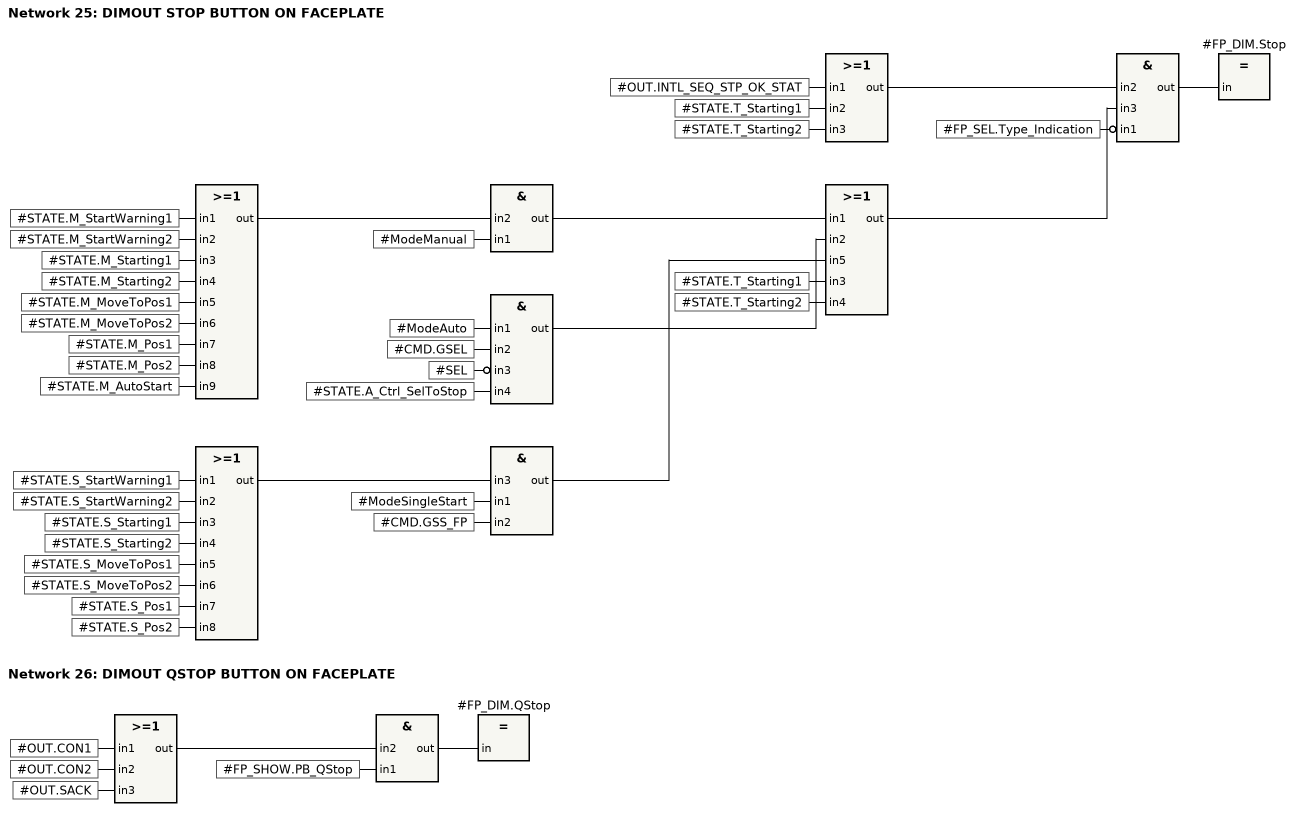
   #FP_DIM.Stop := (#OUT.INTL_SEQ_STP_OK_STAT OR #STATE.T_Starting1 OR #STATE.T_Starting2) AND (((#STATE.M_StartWarning1 OR #STATE.M_StartWarning2 OR #STATE.M_Starting1 OR #STATE.M_Starting2 OR #STATE.M_MoveToPos1 OR #STATE.M_MoveToPos2 OR #STATE.M_Pos1 OR #STATE.M_Pos2 OR #STATE.M_AutoStart) AND #ModeManual) OR (#ModeAuto AND #CMD.GSEL AND NOT #SEL AND #STATE.A_Ctrl_SelToStop) OR ((#STATE.S_StartWarning1 OR #STATE.S_StartWarning2 OR #STATE.S_Starting1 OR #STATE.S_Starting2 OR #STATE.S_MoveToPos1 OR #STATE.S_MoveToPos2 OR #STATE.S_Pos1 OR #STATE.S_Pos2) AND #ModeSingleStart AND #CMD.GSS_FP) OR #STATE.T_Starting1 OR #STATE.T_Starting2) AND NOT #FP_SEL.Type_Indication;
END_REGION

REGION Network 26: DIMOUT QSTOP BUTTON ON FACEPLATE
   #FP_DIM.QStop := (#OUT.CON1 OR #OUT.CON2 OR #OUT.SACK) AND #FP_SHOW.PB_QStop;
END_REGION

REGION Network 27: DIMOUT START1 BUTTON ON FACEPLATE
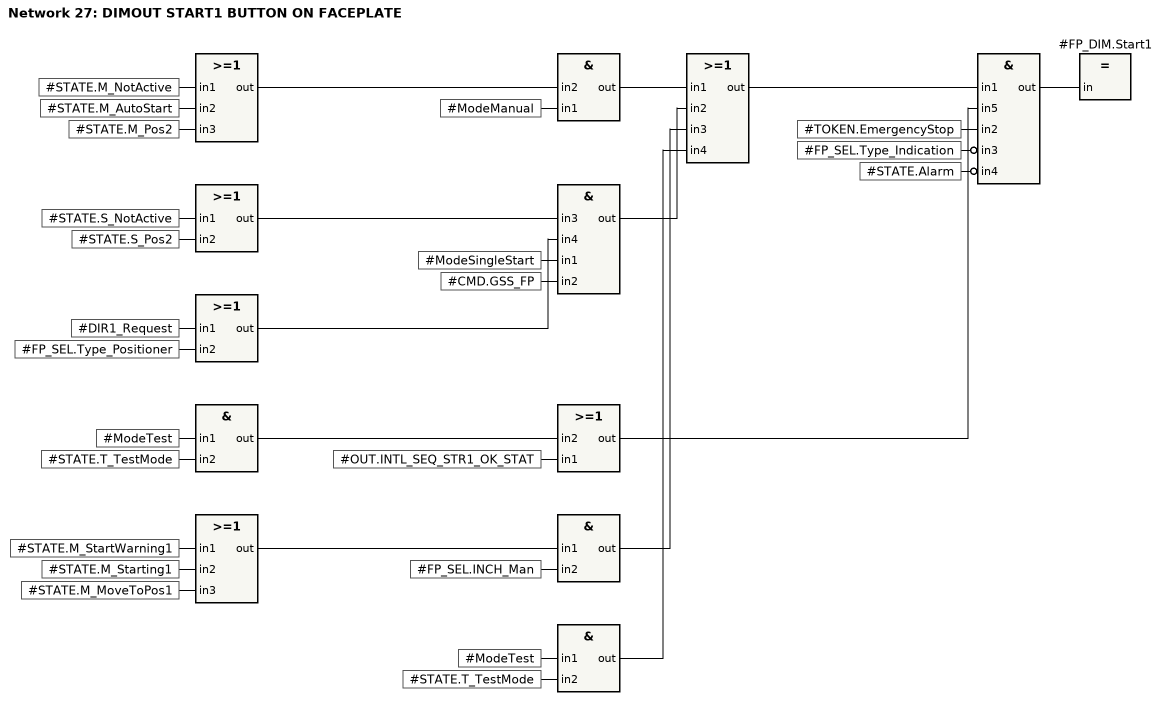
   #FP_DIM.Start1 := (((#STATE.M_NotActive OR #STATE.M_AutoStart OR #STATE.M_Pos2) AND #ModeManual) OR ((#STATE.S_NotActive OR #STATE.S_Pos2) AND (#DIR1_Request OR #FP_SEL.Type_Positioner) AND #ModeSingleStart AND #CMD.GSS_FP) OR ((#STATE.M_StartWarning1 OR #STATE.M_Starting1 OR #STATE.M_MoveToPos1) AND #FP_SEL.INCH_Man) OR (#ModeTest AND #STATE.T_TestMode)) AND ((#ModeTest AND #STATE.T_TestMode) OR #OUT.INTL_SEQ_STR1_OK_STAT) AND #TOKEN.EmergencyStop AND NOT #FP_SEL.Type_Indication AND NOT #STATE.Alarm;
END_REGION

REGION Network 28: DIMOUT START2 BUTTON ON FACEPLATE
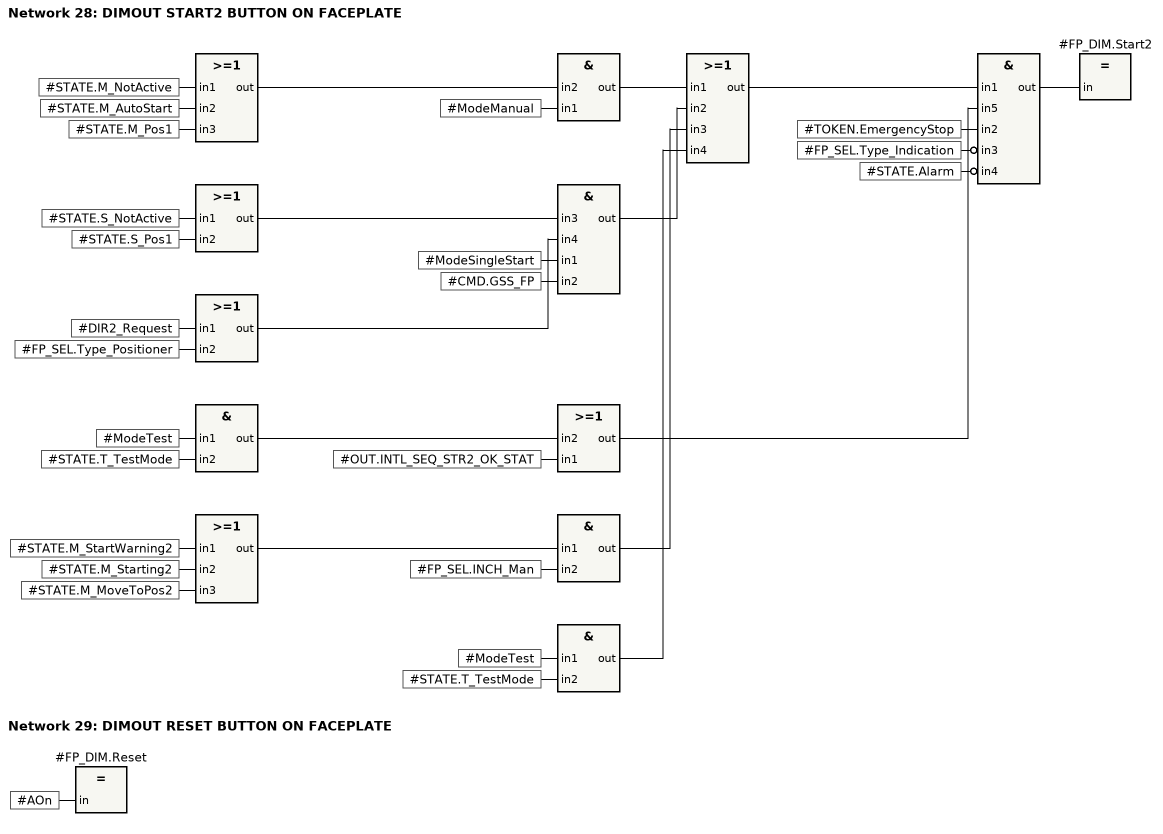
   #FP_DIM.Start2 := (((#STATE.M_NotActive OR #STATE.M_AutoStart OR #STATE.M_Pos1) AND #ModeManual) OR ((#STATE.S_NotActive OR #STATE.S_Pos1) AND (#DIR2_Request OR #FP_SEL.Type_Positioner) AND #ModeSingleStart AND #CMD.GSS_FP) OR ((#STATE.M_StartWarning2 OR #STATE.M_Starting2 OR #STATE.M_MoveToPos2) AND #FP_SEL.INCH_Man) OR (#ModeTest AND #STATE.T_TestMode)) AND ((#ModeTest AND #STATE.T_TestMode) OR #OUT.INTL_SEQ_STR2_OK_STAT) AND #TOKEN.EmergencyStop AND NOT #FP_SEL.Type_Indication AND NOT #STATE.Alarm;
END_REGION

REGION Network 29: DIMOUT RESET BUTTON ON FACEPLATE
   #FP_DIM.Reset := #AOn;
END_REGION

REGION Network 30: Auto Mode
   // Build 002 - 25 March 2019 : REM flag is removed from FP_CMD.Auto condition
   // Build 002 - 25 March 2019 : FP_EN.Mode_Auto flag added to select condition
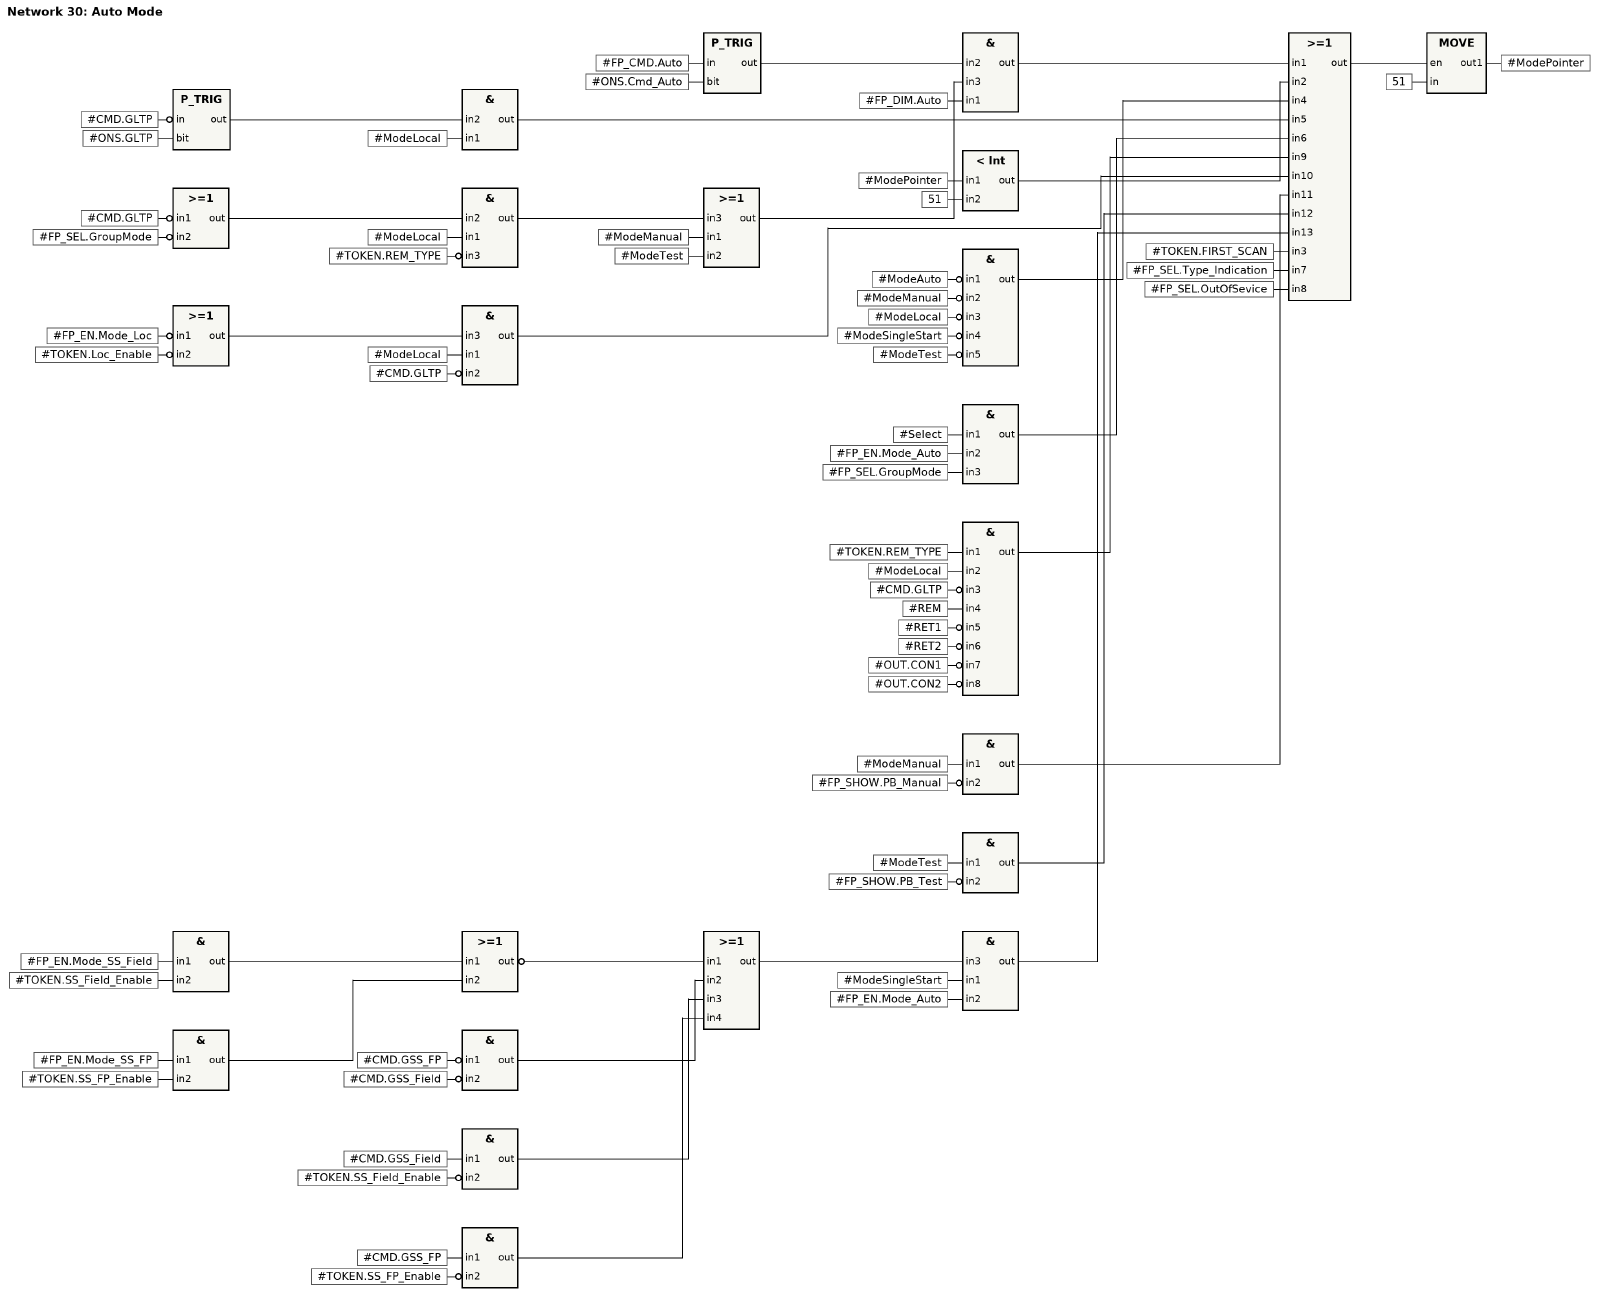
   #_w1 := #FP_CMD.Auto AND NOT #ONS.Cmd_Auto;   // rising edge
   #ONS.Cmd_Auto := #FP_CMD.Auto;
   #_w2 := NOT #CMD.GLTP AND NOT #ONS.GLTP;   // rising edge
   #ONS.GLTP := NOT #CMD.GLTP;
   IF (#_w1 AND (((NOT #CMD.GLTP OR NOT #FP_SEL.GroupMode) AND #ModeLocal AND NOT #TOKEN.REM_TYPE) OR #ModeManual OR #ModeTest) AND #FP_DIM.Auto) OR (#ModePointer < 51) OR (NOT #ModeAuto AND NOT #ModeManual AND NOT #ModeLocal AND NOT #ModeSingleStart AND NOT #ModeTest) OR (#_w2 AND #ModeLocal) OR (#Select AND #FP_EN.Mode_Auto AND #FP_SEL.GroupMode) OR (#TOKEN.REM_TYPE AND #ModeLocal AND NOT #CMD.GLTP AND #REM AND NOT #RET1 AND NOT #RET2 AND NOT #OUT.CON1 AND NOT #OUT.CON2) OR ((NOT #FP_EN.Mode_Loc OR NOT #TOKEN.Loc_Enable) AND #ModeLocal AND NOT #CMD.GLTP) OR (#ModeManual AND NOT #FP_SHOW.PB_Manual) OR (#ModeTest AND NOT #FP_SHOW.PB_Test) OR ((NOT ((#FP_EN.Mode_SS_Field AND #TOKEN.SS_Field_Enable) OR (#FP_EN.Mode_SS_FP AND #TOKEN.SS_FP_Enable)) OR (NOT #CMD.GSS_FP AND NOT #CMD.GSS_Field) OR (#CMD.GSS_Field AND NOT #TOKEN.SS_Field_Enable) OR (#CMD.GSS_FP AND NOT #TOKEN.SS_FP_Enable)) AND #ModeSingleStart AND #FP_EN.Mode_Auto) OR #TOKEN.FIRST_SCAN OR #FP_SEL.Type_Indication OR #FP_SEL.OutOfSevice THEN
       #ModePointer := 51;
   END_IF;
END_REGION

REGION Network 31: Mode Manual
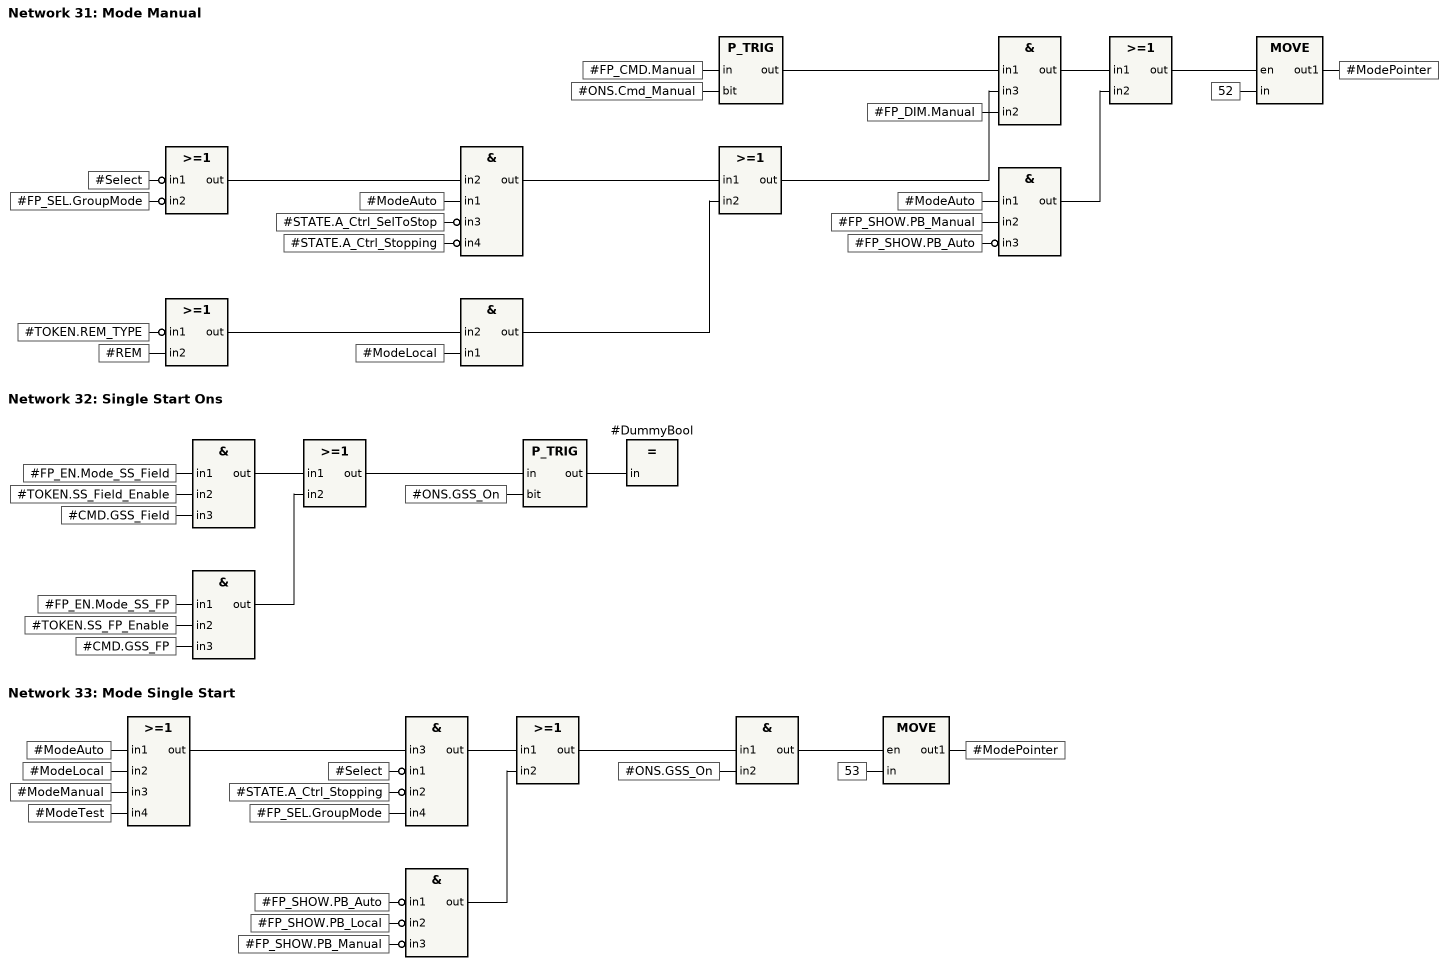
   #_w1 := #FP_CMD.Manual AND NOT #ONS.Cmd_Manual;   // rising edge
   #ONS.Cmd_Manual := #FP_CMD.Manual;
   IF (#_w1 AND (((NOT #Select OR NOT #FP_SEL.GroupMode) AND #ModeAuto AND NOT #STATE.A_Ctrl_SelToStop AND NOT #STATE.A_Ctrl_Stopping) OR ((NOT #TOKEN.REM_TYPE OR #REM) AND #ModeLocal)) AND #FP_DIM.Manual) OR (#ModeAuto AND #FP_SHOW.PB_Manual AND NOT #FP_SHOW.PB_Auto) THEN
       #ModePointer := 52;
   END_IF;
END_REGION

REGION Network 32: Single Start Ons
   // Build 003 - 2.July.2019 (EXTBOB): Added ONS and Created New Network to separate trigger from pre-conditions
   #_w1 := (#FP_EN.Mode_SS_Field AND #TOKEN.SS_Field_Enable AND #CMD.GSS_Field) OR (#FP_EN.Mode_SS_FP AND #TOKEN.SS_FP_Enable AND #CMD.GSS_FP);
   #_w2 := #_w1 AND NOT #ONS.GSS_On;   // rising edge
   #ONS.GSS_On := #_w1;
   #DummyBool := #_w2;
END_REGION

REGION Network 33: Mode Single Start
   // Build 003 - 2.July.2019 (EXTBOB): Added Single Start ONS and Removed the Single start trigger condition & made as seperate Network above
   IF (((#ModeAuto OR #ModeLocal OR #ModeManual OR #ModeTest) AND NOT #Select AND NOT #STATE.A_Ctrl_Stopping AND #FP_SEL.GroupMode) OR (NOT #FP_SHOW.PB_Auto AND NOT #FP_SHOW.PB_Local AND NOT #FP_SHOW.PB_Manual)) AND #ONS.GSS_On THEN
       #ModePointer := 53;
   END_IF;
END_REGION

REGION Network 34: Mode Local
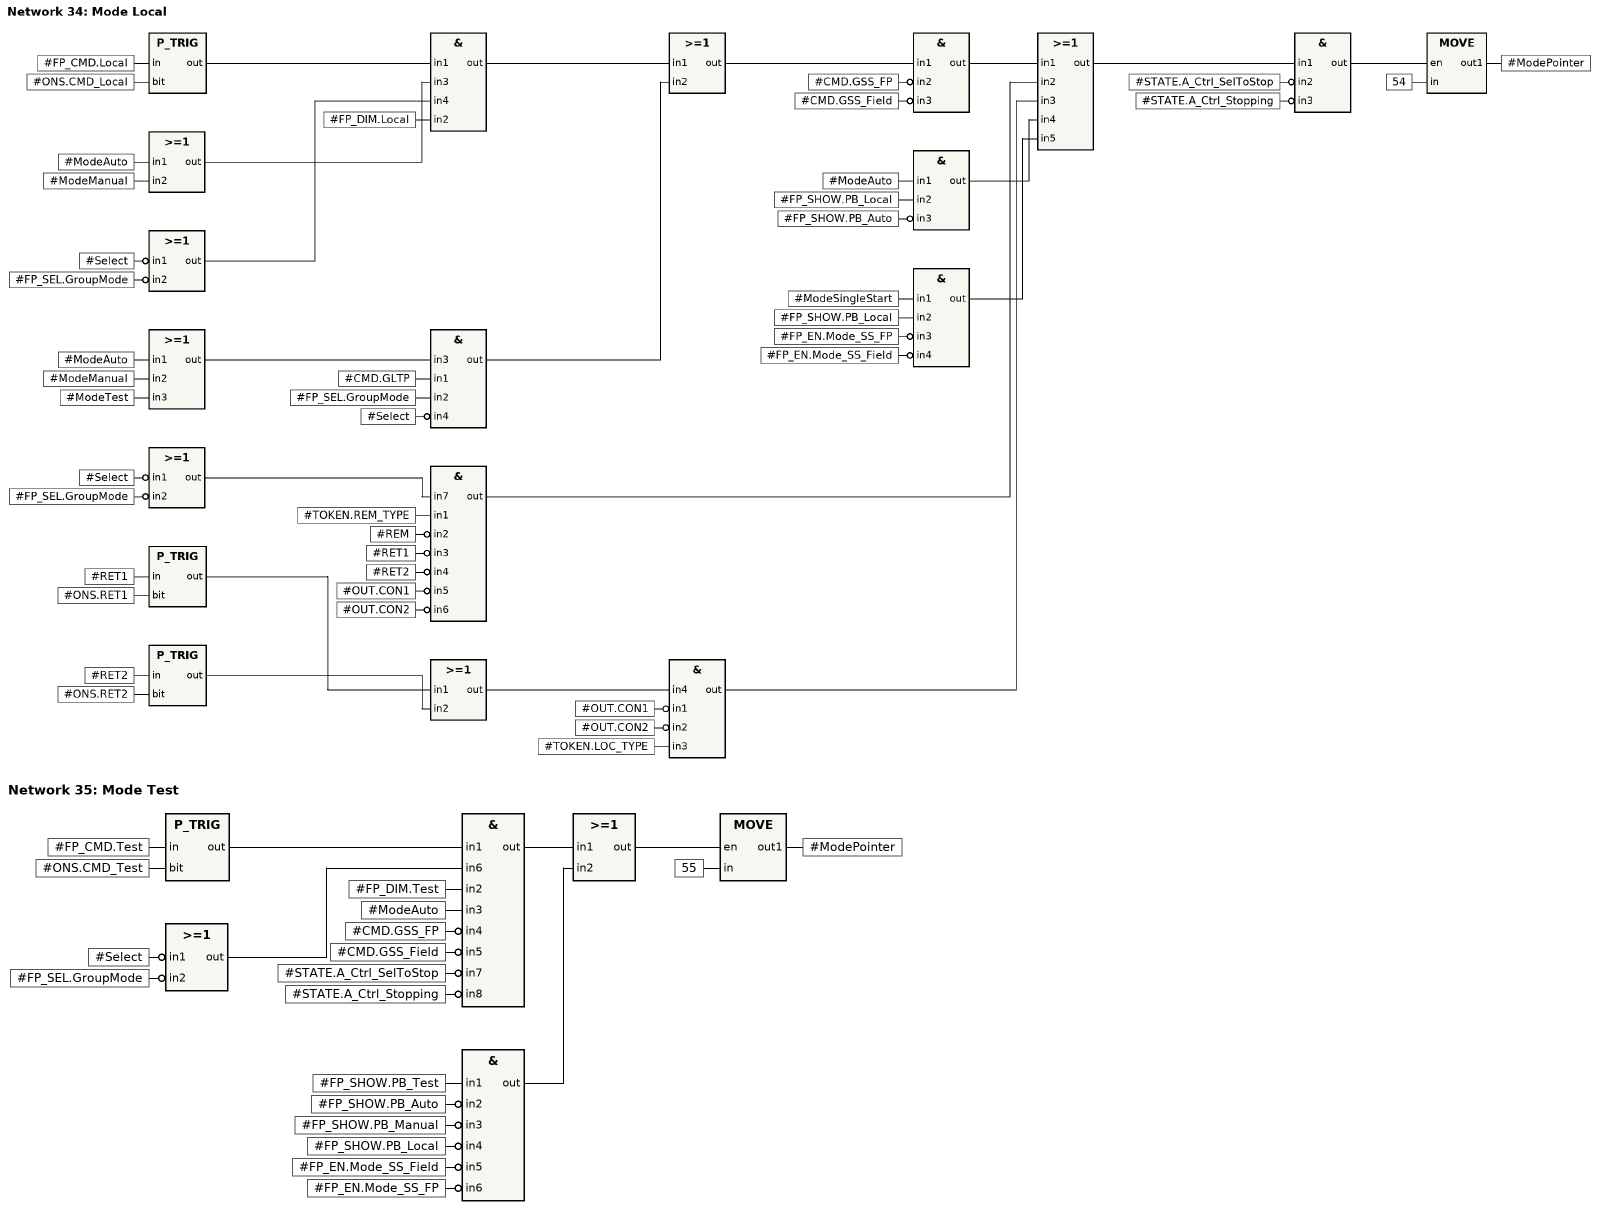
   #_w1 := #FP_CMD.Local AND NOT #ONS.CMD_Local;   // rising edge
   #ONS.CMD_Local := #FP_CMD.Local;
   #_w2 := #RET1 AND NOT #ONS.RET1;   // rising edge
   #ONS.RET1 := #RET1;
   #_w3 := #RET2 AND NOT #ONS.RET2;   // rising edge
   #ONS.RET2 := #RET2;
   IF ((((#_w1 AND (#ModeAuto OR #ModeManual) AND (NOT #Select OR NOT #FP_SEL.GroupMode) AND #FP_DIM.Local) OR ((#ModeAuto OR #ModeManual OR #ModeTest) AND #CMD.GLTP AND #FP_SEL.GroupMode AND NOT #Select)) AND NOT #CMD.GSS_FP AND NOT #CMD.GSS_Field) OR ((NOT #Select OR NOT #FP_SEL.GroupMode) AND #TOKEN.REM_TYPE AND NOT #REM AND NOT #RET1 AND NOT #RET2 AND NOT #OUT.CON1 AND NOT #OUT.CON2) OR ((#_w2 OR #_w3) AND NOT #OUT.CON1 AND NOT #OUT.CON2 AND #TOKEN.LOC_TYPE) OR (#ModeAuto AND #FP_SHOW.PB_Local AND NOT #FP_SHOW.PB_Auto) OR (#ModeSingleStart AND #FP_SHOW.PB_Local AND NOT #FP_EN.Mode_SS_FP AND NOT #FP_EN.Mode_SS_Field)) AND NOT #STATE.A_Ctrl_SelToStop AND NOT #STATE.A_Ctrl_Stopping THEN
       #ModePointer := 54;
   END_IF;
END_REGION

REGION Network 35: Mode Test
   #_w1 := #FP_CMD.Test AND NOT #ONS.CMD_Test;   // rising edge
   #ONS.CMD_Test := #FP_CMD.Test;
   IF (#_w1 AND (NOT #Select OR NOT #FP_SEL.GroupMode) AND #FP_DIM.Test AND #ModeAuto AND NOT #CMD.GSS_FP AND NOT #CMD.GSS_Field AND NOT #STATE.A_Ctrl_SelToStop AND NOT #STATE.A_Ctrl_Stopping) OR (#FP_SHOW.PB_Test AND NOT #FP_SHOW.PB_Auto AND NOT #FP_SHOW.PB_Manual AND NOT #FP_SHOW.PB_Local AND NOT #FP_EN.Mode_SS_Field AND NOT #FP_EN.Mode_SS_FP) THEN
       #ModePointer := 55;
   END_IF;
END_REGION

REGION Network 36: Mode Auto
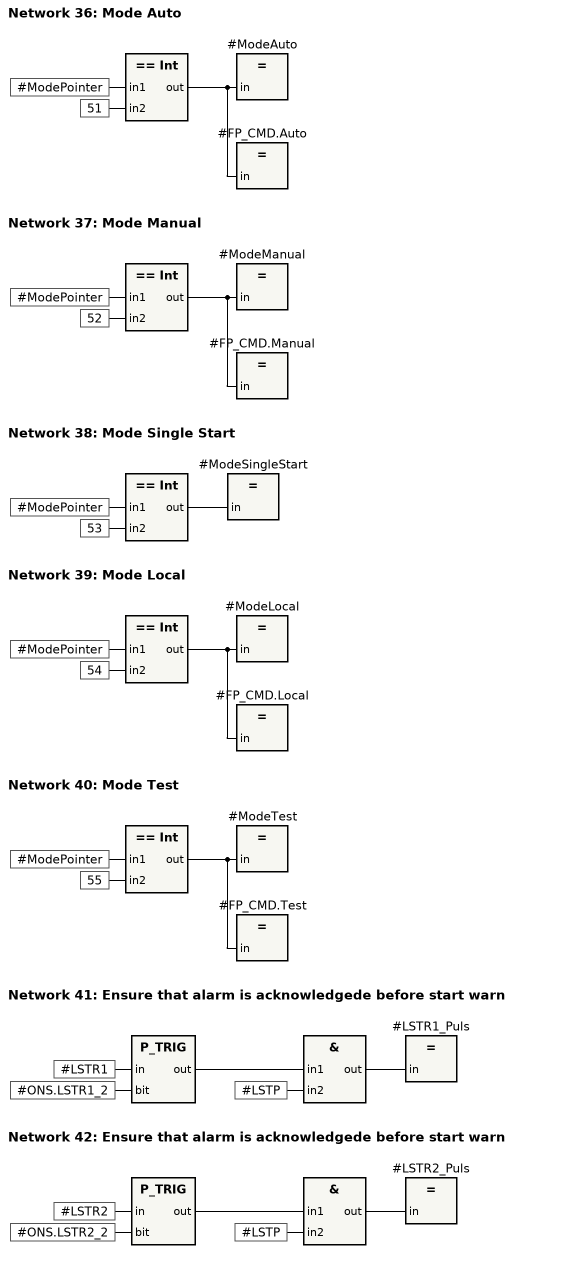
   #ModeAuto := #ModePointer = 51;
   #FP_CMD.Auto := #ModeAuto;
END_REGION

REGION Network 37: Mode Manual
   #ModeManual := #ModePointer = 52;
   #FP_CMD.Manual := #ModeManual;
END_REGION

REGION Network 38: Mode Single Start
   #ModeSingleStart := #ModePointer = 53;
END_REGION

REGION Network 39: Mode Local
   #ModeLocal := #ModePointer = 54;
   #FP_CMD.Local := #ModeLocal;
END_REGION

REGION Network 40: Mode Test
   #ModeTest := #ModePointer = 55;
   #FP_CMD.Test := #ModeTest;
END_REGION

REGION Network 41: Ensure that alarm is acknowledgede before start warn
   // Build 003 - 30 June 2019 (EXTBOB): Added LSTP to prevent pulse output
   #_w1 := #LSTR1 AND NOT #ONS.LSTR1_2;   // rising edge
   #ONS.LSTR1_2 := #LSTR1;
   #LSTR1_Puls := #_w1 AND #LSTP;
END_REGION

REGION Network 42: Ensure that alarm is acknowledgede before start warn
   // Build 003 - 30 June 2019 (EXTBOB): Added LSTP to prevent pulse output
   #_w1 := #LSTR2 AND NOT #ONS.LSTR2_2;   // rising edge
   #ONS.LSTR2_2 := #LSTR2;
   #LSTR2_Puls := #_w1 AND #LSTP;
END_REGION

REGION Network 43: FACEPLATE COMMANDS (Pulse Type)
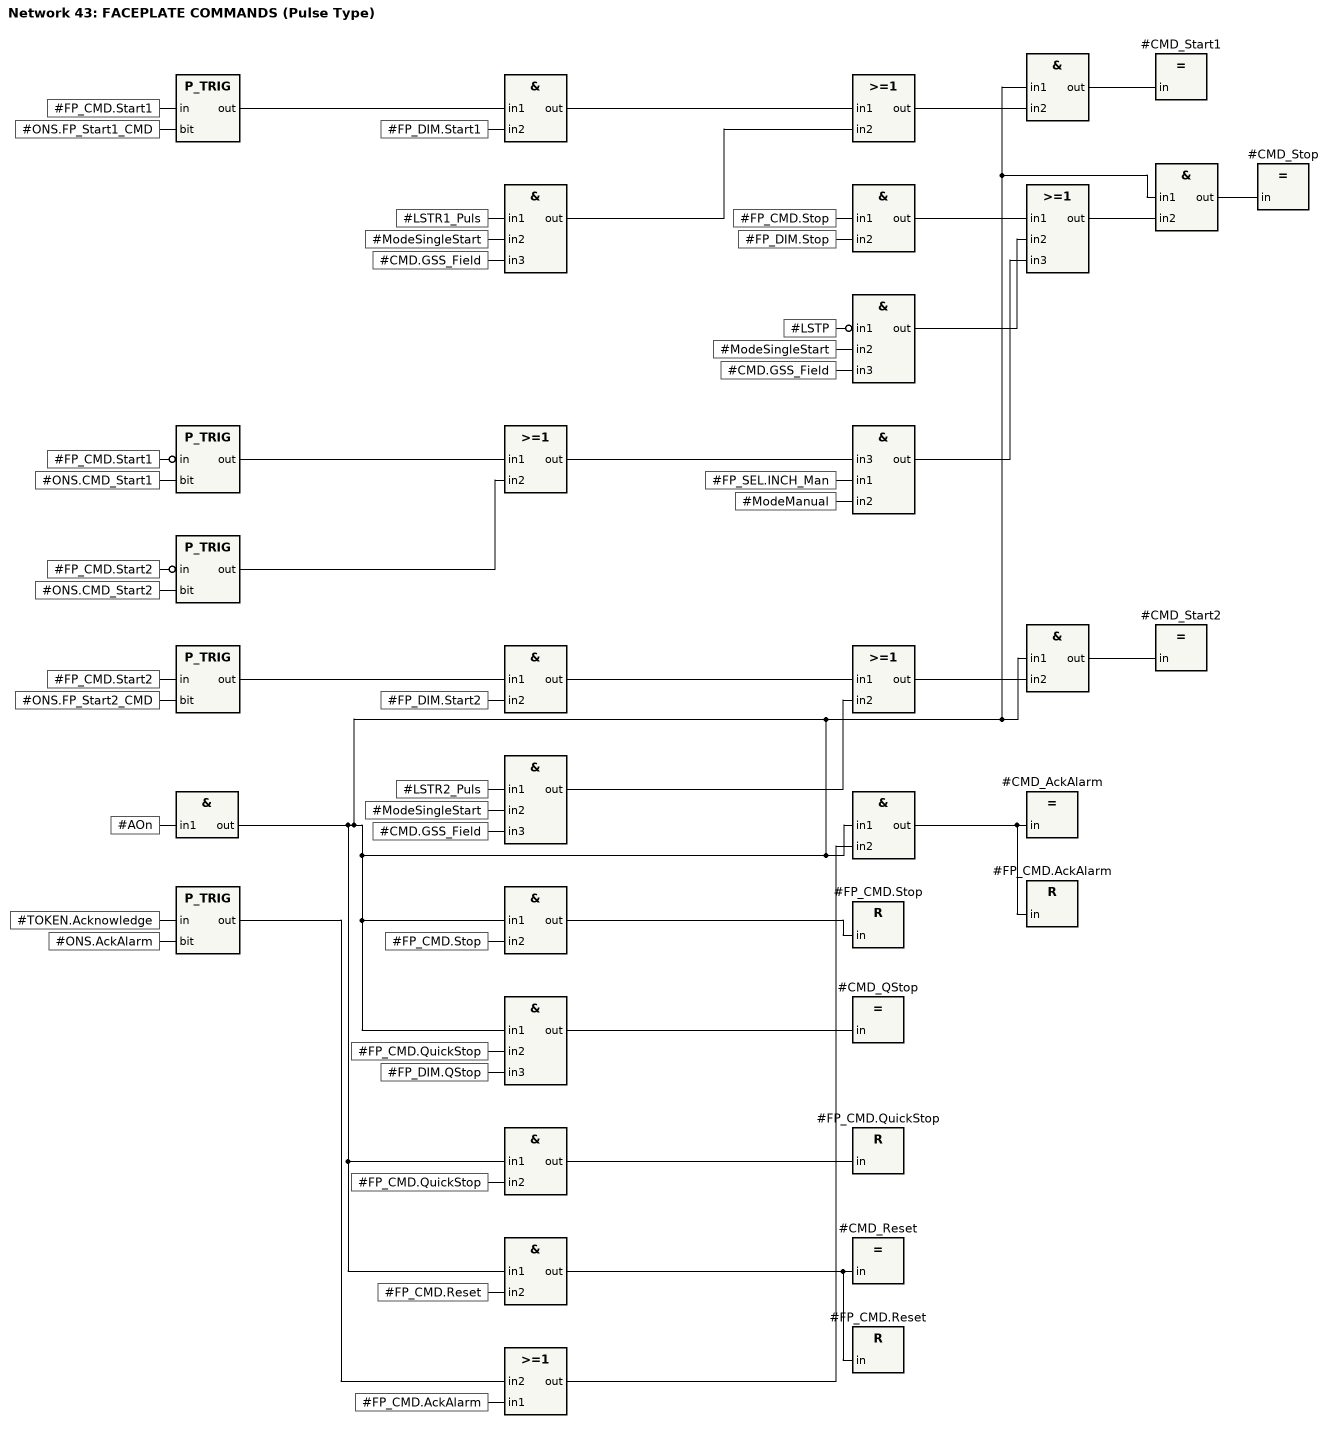
   #_w1 := #FP_CMD.Start1 AND NOT #ONS.FP_Start1_CMD;   // rising edge
   #ONS.FP_Start1_CMD := #FP_CMD.Start1;
   #CMD_Start1 := #AOn AND ((#_w1 AND #FP_DIM.Start1) OR (#LSTR1_Puls AND #ModeSingleStart AND #CMD.GSS_Field));
   #_w2 := #FP_CMD.Start2 AND NOT #ONS.FP_Start2_CMD;   // rising edge
   #ONS.FP_Start2_CMD := #FP_CMD.Start2;
   #CMD_Start2 := #AOn AND ((#_w2 AND #FP_DIM.Start2) OR (#LSTR2_Puls AND #ModeSingleStart AND #CMD.GSS_Field));
   #_w3 := NOT #FP_CMD.Start1 AND NOT #ONS.CMD_Start1;   // rising edge
   #ONS.CMD_Start1 := NOT #FP_CMD.Start1;
   #_w4 := NOT #FP_CMD.Start2 AND NOT #ONS.CMD_Start2;   // rising edge
   #ONS.CMD_Start2 := NOT #FP_CMD.Start2;
   #CMD_Stop := #AOn AND ((#FP_CMD.Stop AND #FP_DIM.Stop) OR (NOT #LSTP AND #ModeSingleStart AND #CMD.GSS_Field) OR ((#_w3 OR #_w4) AND #FP_SEL.INCH_Man AND #ModeManual));
   IF #AOn AND #FP_CMD.Stop THEN #FP_CMD.Stop := FALSE; END_IF;
   #CMD_QStop := #AOn AND #FP_CMD.QuickStop AND #FP_DIM.QStop;
   IF #AOn AND #FP_CMD.QuickStop THEN #FP_CMD.QuickStop := FALSE; END_IF;
   #CMD_Reset := #AOn AND #FP_CMD.Reset;
   IF #CMD_Reset THEN #FP_CMD.Reset := FALSE; END_IF;
   #_w5 := #TOKEN.Acknowledge AND NOT #ONS.AckAlarm;   // rising edge
   #ONS.AckAlarm := #TOKEN.Acknowledge;
   #CMD_AckAlarm := #AOn AND (#_w5 OR #FP_CMD.AckAlarm);
   IF #CMD_AckAlarm THEN #FP_CMD.AckAlarm := FALSE; END_IF;
END_REGION

REGION Network 44: FACEPLATE COMMANDS (Pulse Type)
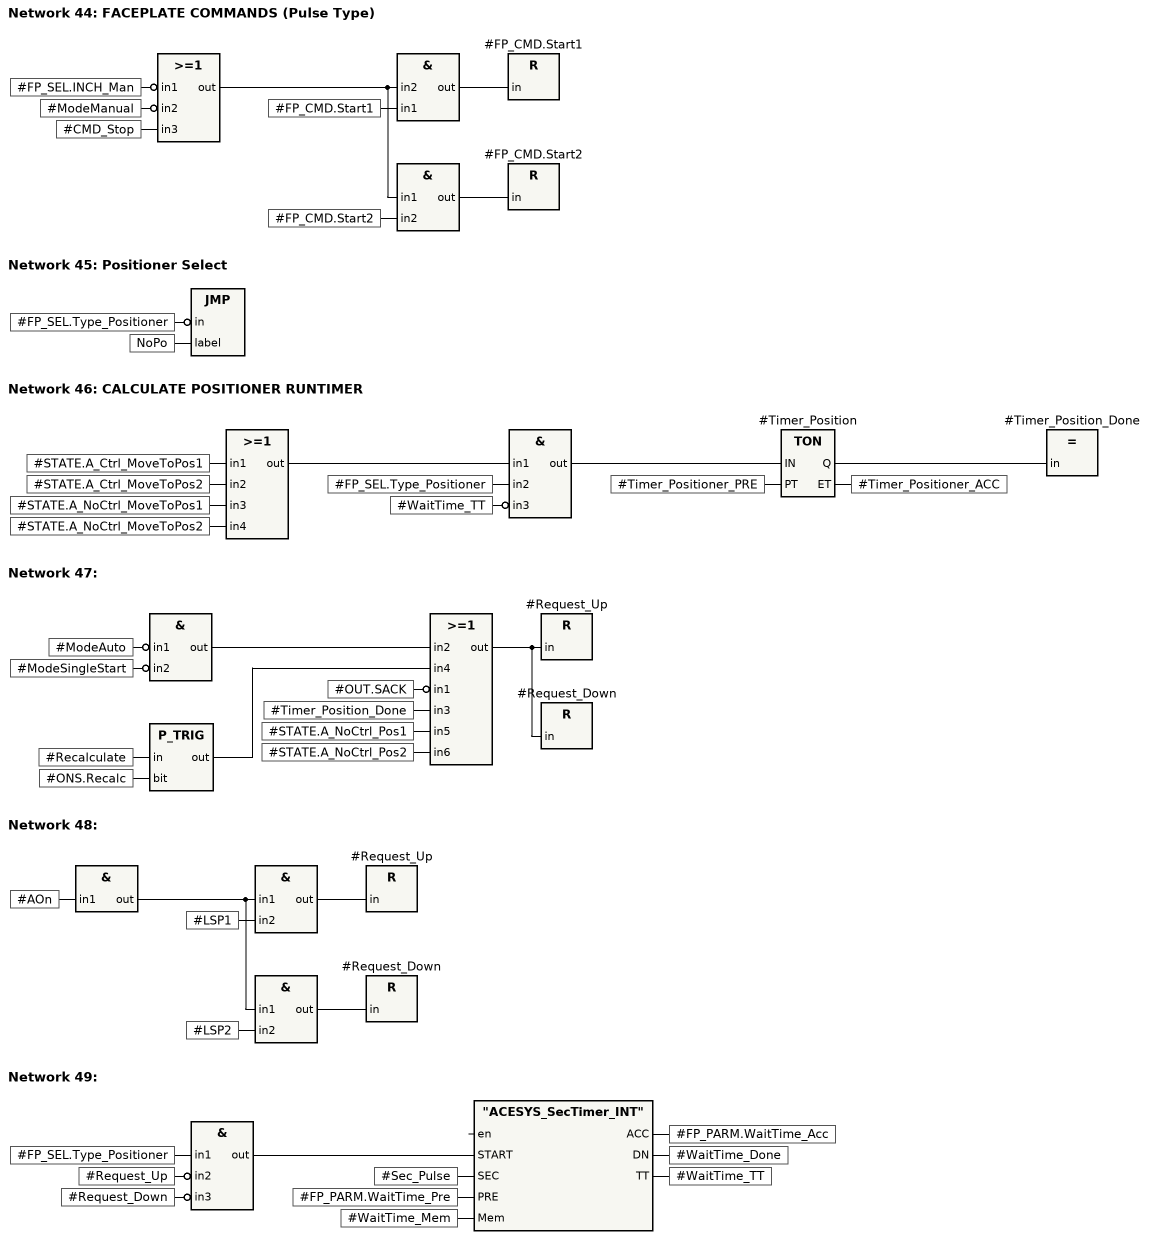
   #_w1 := NOT #FP_SEL.INCH_Man OR NOT #ModeManual OR #CMD_Stop;
   IF #_w1 AND #FP_CMD.Start1 THEN #FP_CMD.Start1 := FALSE; END_IF;
   IF #_w1 AND #FP_CMD.Start2 THEN #FP_CMD.Start2 := FALSE; END_IF;
END_REGION

REGION Network 45: Positioner Select
   IF NOT #FP_SEL.Type_Positioner THEN GOTO NoPo; END_IF;
END_REGION

REGION Network 46: CALCULATE POSITIONER RUNTIMER
   #Timer_Position(IN := (#STATE.A_Ctrl_MoveToPos1 OR #STATE.A_Ctrl_MoveToPos2 OR #STATE.A_NoCtrl_MoveToPos1 OR #STATE.A_NoCtrl_MoveToPos2) AND #FP_SEL.Type_Positioner AND NOT #WaitTime_TT,   // TON
                   PT := #Timer_Positioner_PRE,
                   ET => #Timer_Positioner_ACC);
   #Timer_Position_Done := #Timer_Position.Q;
END_REGION

REGION Network 47
   #_w1 := #Recalculate AND NOT #ONS.Recalc;   // rising edge
   #ONS.Recalc := #Recalculate;
   IF (NOT #ModeAuto AND NOT #ModeSingleStart) OR #_w1 OR NOT #OUT.SACK OR #Timer_Position_Done OR #STATE.A_NoCtrl_Pos1 OR #STATE.A_NoCtrl_Pos2 THEN
       #Request_Up := FALSE;
       #Request_Down := FALSE;
   END_IF;
END_REGION

REGION Network 48
   IF #AOn AND #LSP1 THEN #Request_Up := FALSE; END_IF;
   IF #AOn AND #LSP2 THEN #Request_Down := FALSE; END_IF;
END_REGION

REGION Network 49
   "ACESYS_SecTimer_INT"(START := #FP_SEL.Type_Positioner AND NOT #Request_Up AND NOT #Request_Down,
                         SEC := #Sec_Pulse,
                         PRE := #FP_PARM.WaitTime_Pre,
                         Mem := #WaitTime_Mem,
                         ACC => #FP_PARM.WaitTime_Acc,
                         DN => #WaitTime_Done,
                         TT => #WaitTime_TT);
END_REGION

REGION Network 50
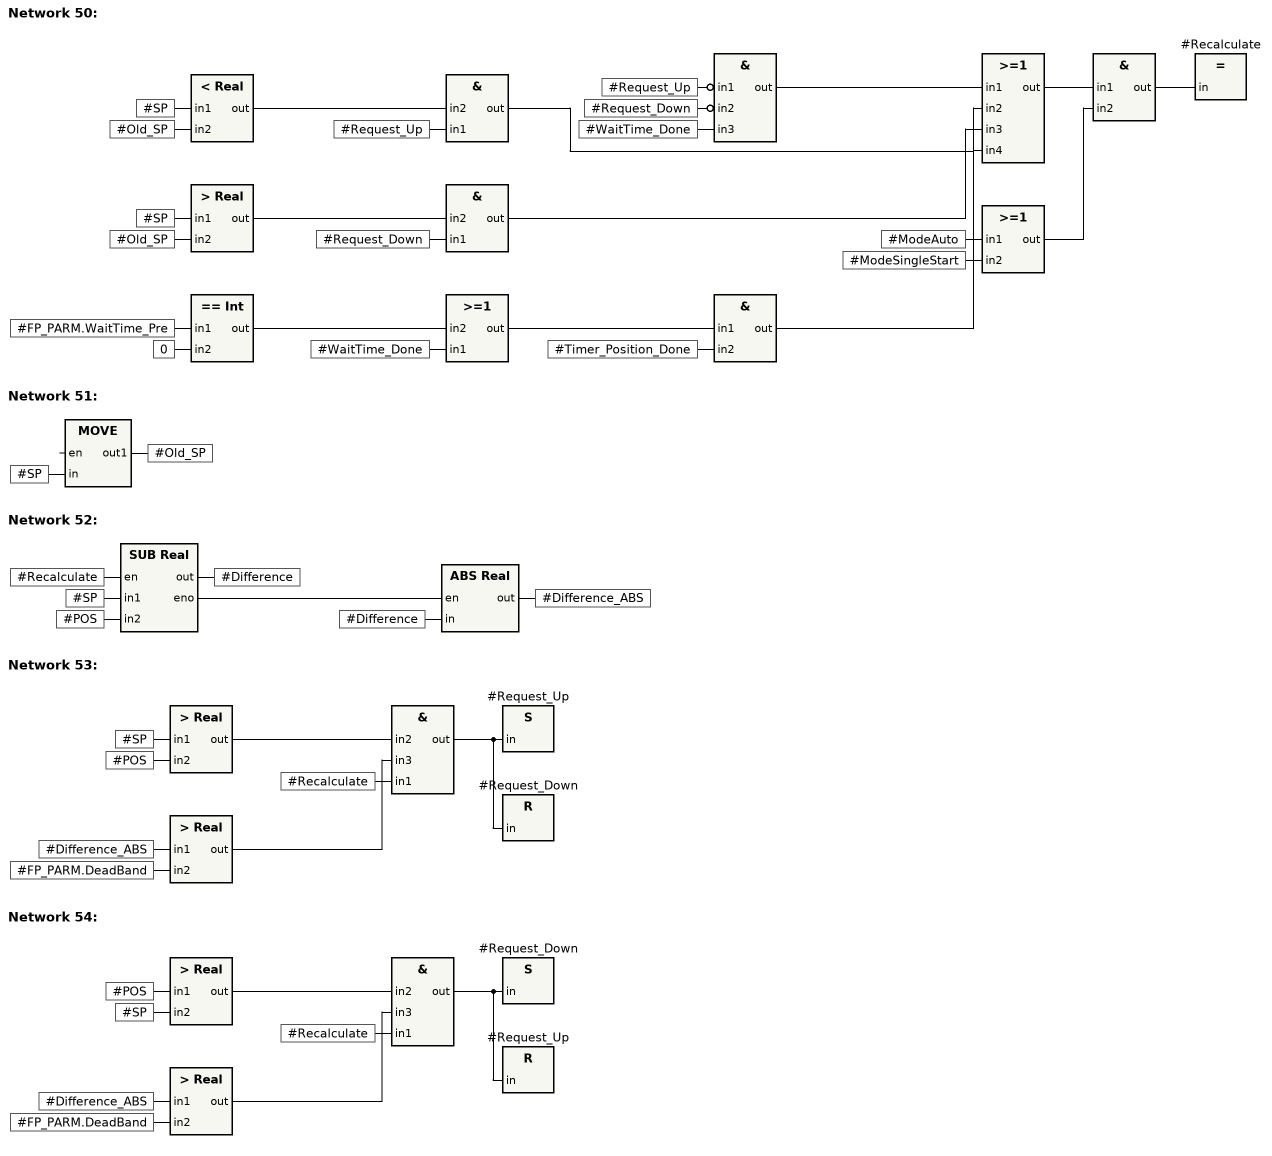
   #Recalculate := ((NOT #Request_Up AND NOT #Request_Down AND #WaitTime_Done) OR ((#SP < #Old_SP) AND #Request_Up) OR ((#SP > #Old_SP) AND #Request_Down) OR (((#FP_PARM.WaitTime_Pre = 0) OR #WaitTime_Done) AND #Timer_Position_Done)) AND (#ModeAuto OR #ModeSingleStart);
END_REGION

REGION Network 51
   #Old_SP := #SP;
END_REGION

REGION Network 52
   // ENO of a box is taken as its EN; it also drops when the box reports an error
   IF #Recalculate THEN
       #Difference := #SP - #POS;
       #Difference_ABS := ABS(#Difference);
   END_IF;
END_REGION

REGION Network 53
   IF (#SP > #POS) AND (#Difference_ABS > #FP_PARM.DeadBand) AND #Recalculate THEN
       #Request_Up := TRUE;
       #Request_Down := FALSE;
   END_IF;
END_REGION

REGION Network 54
   IF (#POS > #SP) AND (#Difference_ABS > #FP_PARM.DeadBand) AND #Recalculate THEN
       #Request_Down := TRUE;
       #Request_Up := FALSE;
   END_IF;
END_REGION

REGION Network 55
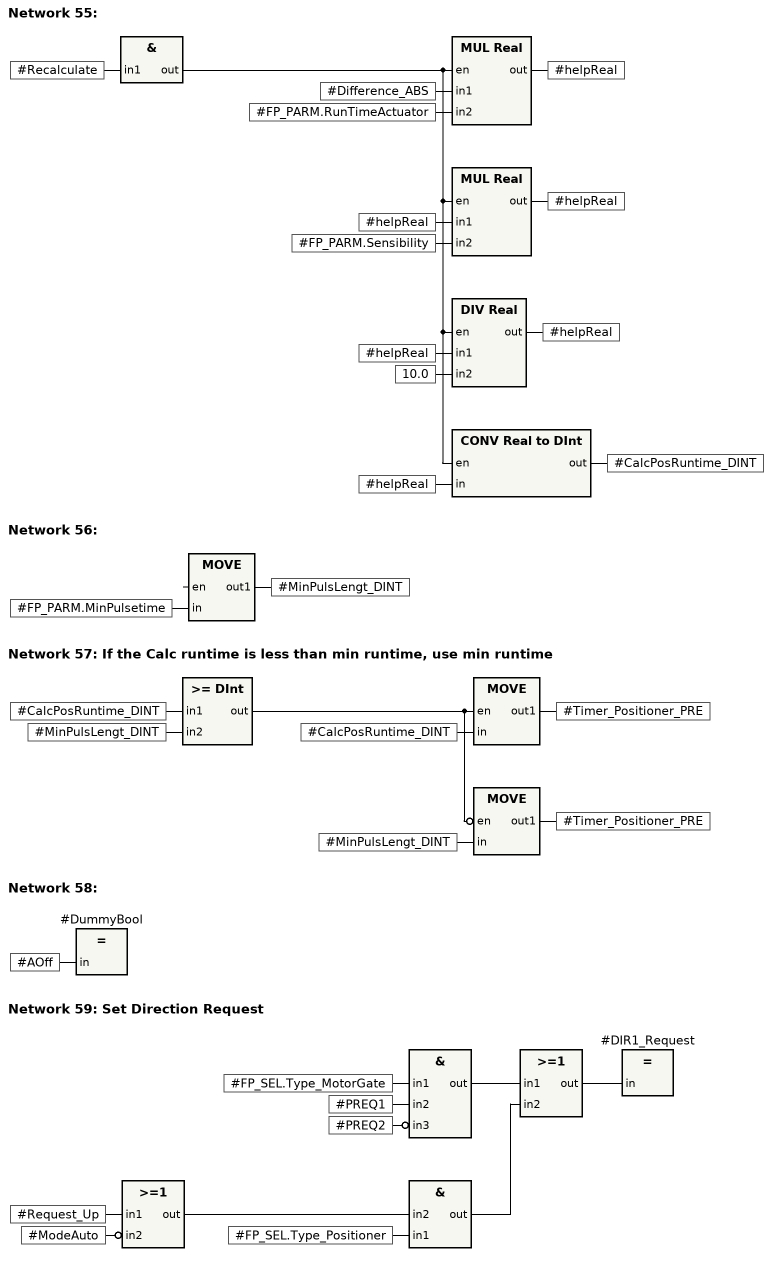
   IF #Recalculate THEN
       #helpReal := #Difference_ABS * #FP_PARM.RunTimeActuator;
       #helpReal := #helpReal * #FP_PARM.Sensibility;
       #helpReal := #helpReal / 10.0;
       #CalcPosRuntime_DINT := REAL_TO_DINT(#helpReal);
   END_IF;
END_REGION

REGION Network 56
   #MinPulsLengt_DINT := #FP_PARM.MinPulsetime;
END_REGION

REGION Network 57: If the Calc runtime is less than min runtime, use min runtime
   #_w1 := #CalcPosRuntime_DINT >= #MinPulsLengt_DINT;
   IF #_w1 THEN #Timer_Positioner_PRE := #CalcPosRuntime_DINT; END_IF;
   IF NOT #_w1 THEN #Timer_Positioner_PRE := #MinPulsLengt_DINT; END_IF;
END_REGION

REGION Network 58
   NoPo:
   #DummyBool := #AOff;
END_REGION

REGION Network 59: Set Direction Request
   #DIR1_Request := (#FP_SEL.Type_MotorGate AND #PREQ1 AND NOT #PREQ2) OR ((#Request_Up OR NOT #ModeAuto) AND #FP_SEL.Type_Positioner);
END_REGION

REGION Network 60
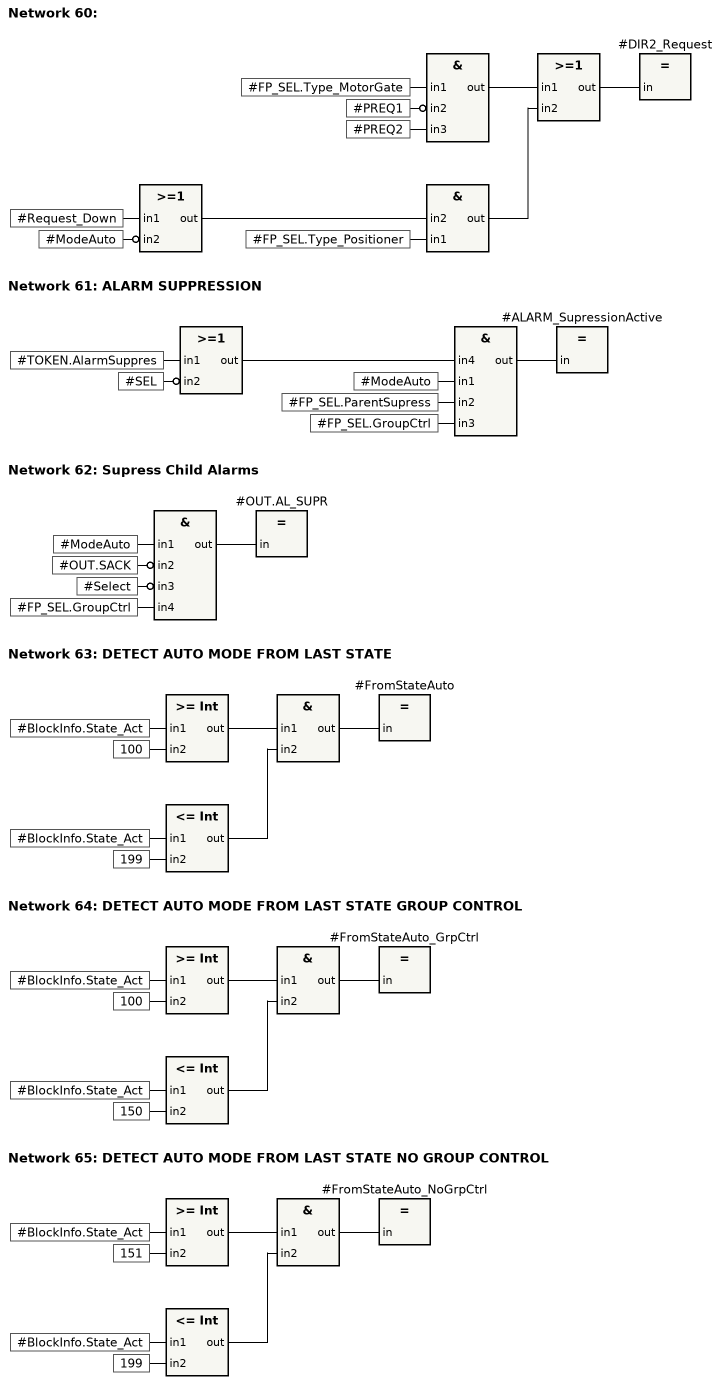
   #DIR2_Request := (#FP_SEL.Type_MotorGate AND NOT #PREQ1 AND #PREQ2) OR ((#Request_Down OR NOT #ModeAuto) AND #FP_SEL.Type_Positioner);
END_REGION

REGION Network 61: ALARM SUPPRESSION
   #ALARM_SupressionActive := (#TOKEN.AlarmSuppres OR NOT #SEL) AND #ModeAuto AND #FP_SEL.ParentSupress AND #FP_SEL.GroupCtrl;
END_REGION

REGION Network 62: Supress Child Alarms
   #OUT.AL_SUPR := #ModeAuto AND NOT #OUT.SACK AND NOT #Select AND #FP_SEL.GroupCtrl;
END_REGION

REGION Network 63: DETECT AUTO MODE FROM LAST STATE
   #FromStateAuto := (#BlockInfo.State_Act >= 100) AND (#BlockInfo.State_Act <= 199);
END_REGION

REGION Network 64: DETECT AUTO MODE FROM LAST STATE GROUP CONTROL
   #FromStateAuto_GrpCtrl := (#BlockInfo.State_Act >= 100) AND (#BlockInfo.State_Act <= 150);
END_REGION

REGION Network 65: DETECT AUTO MODE FROM LAST STATE NO GROUP CONTROL
   #FromStateAuto_NoGrpCtrl := (#BlockInfo.State_Act >= 151) AND (#BlockInfo.State_Act <= 199);
END_REGION

REGION Network 66: DETECT SS MODE FROM LAST STATE
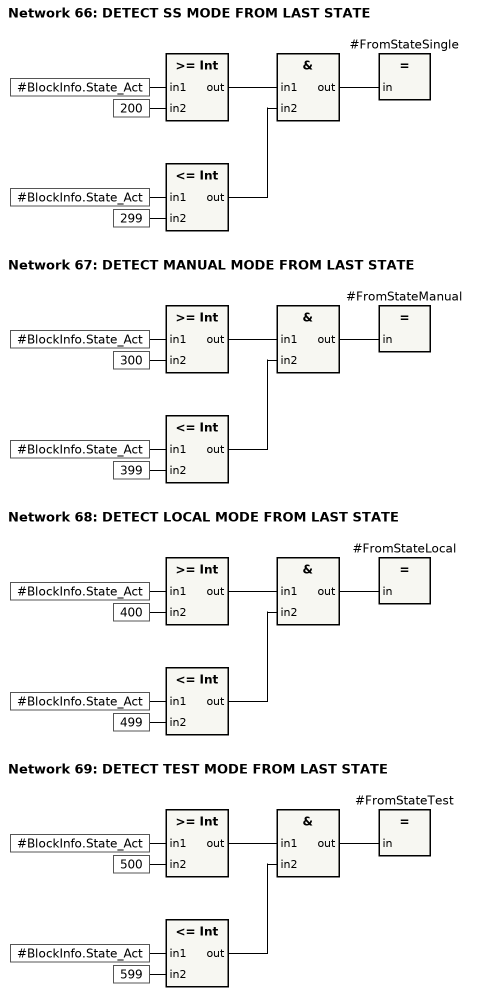
   #FromStateSingle := (#BlockInfo.State_Act >= 200) AND (#BlockInfo.State_Act <= 299);
END_REGION

REGION Network 67: DETECT MANUAL MODE FROM LAST STATE
   #FromStateManual := (#BlockInfo.State_Act >= 300) AND (#BlockInfo.State_Act <= 399);
END_REGION

REGION Network 68: DETECT LOCAL MODE FROM LAST STATE
   #FromStateLocal := (#BlockInfo.State_Act >= 400) AND (#BlockInfo.State_Act <= 499);
END_REGION

REGION Network 69: DETECT TEST MODE FROM LAST STATE
   #FromStateTest := (#BlockInfo.State_Act >= 500) AND (#BlockInfo.State_Act <= 599);
END_REGION

REGION Network 70: DETECT MODE FROM LAST STATE - STOP STATE
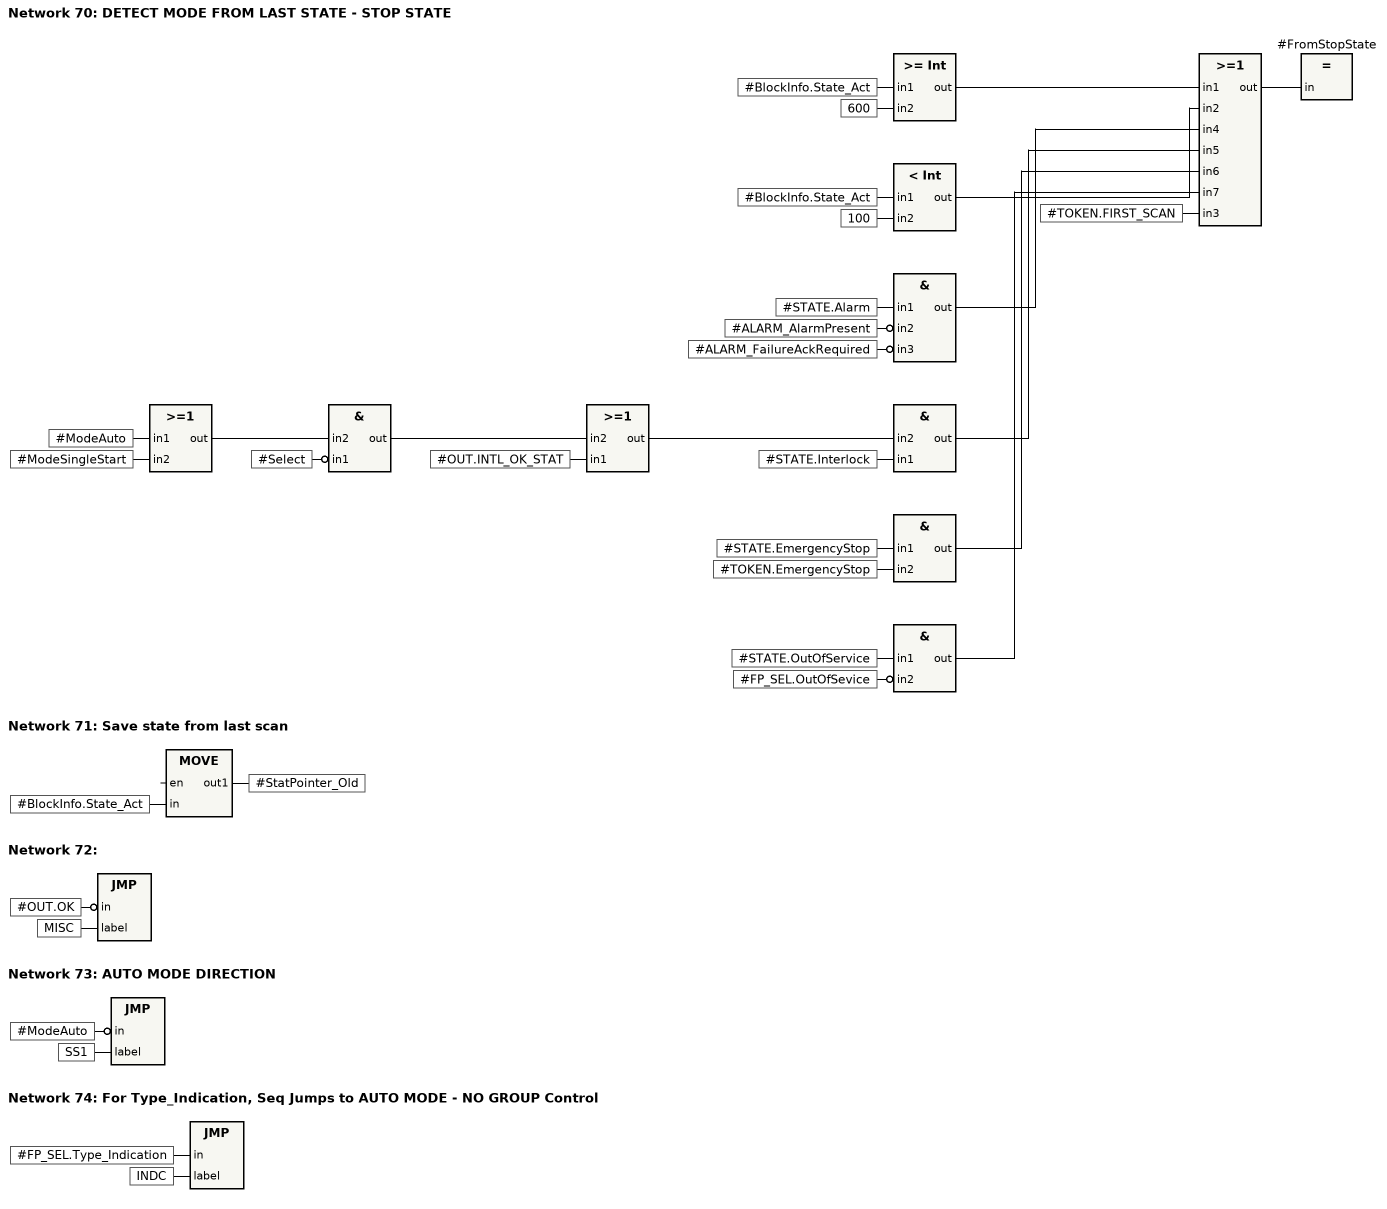
   #FromStopState := (#BlockInfo.State_Act >= 600) OR (#BlockInfo.State_Act < 100) OR (#STATE.Alarm AND NOT #ALARM_AlarmPresent AND NOT #ALARM_FailureAckRequired) OR ((((#ModeAuto OR #ModeSingleStart) AND NOT #Select) OR #OUT.INTL_OK_STAT) AND #STATE.Interlock) OR (#STATE.EmergencyStop AND #TOKEN.EmergencyStop) OR (#STATE.OutOfService AND NOT #FP_SEL.OutOfSevice) OR #TOKEN.FIRST_SCAN;
END_REGION

REGION Network 71: Save state from last scan
   #StatPointer_Old := #BlockInfo.State_Act;
END_REGION

REGION Network 72
   IF NOT #OUT.OK THEN GOTO MISC; END_IF;
END_REGION

REGION Network 73: AUTO MODE DIRECTION
   IF NOT #ModeAuto THEN GOTO SS1; END_IF;
END_REGION

REGION Network 74: For Type_Indication, Seq Jumps to AUTO MODE - NO GROUP Control
   IF #FP_SEL.Type_Indication THEN GOTO INDC; END_IF;
END_REGION

REGION Network 75: AUTO MODE - GROUP CONTROL - State: Auto - Stopped
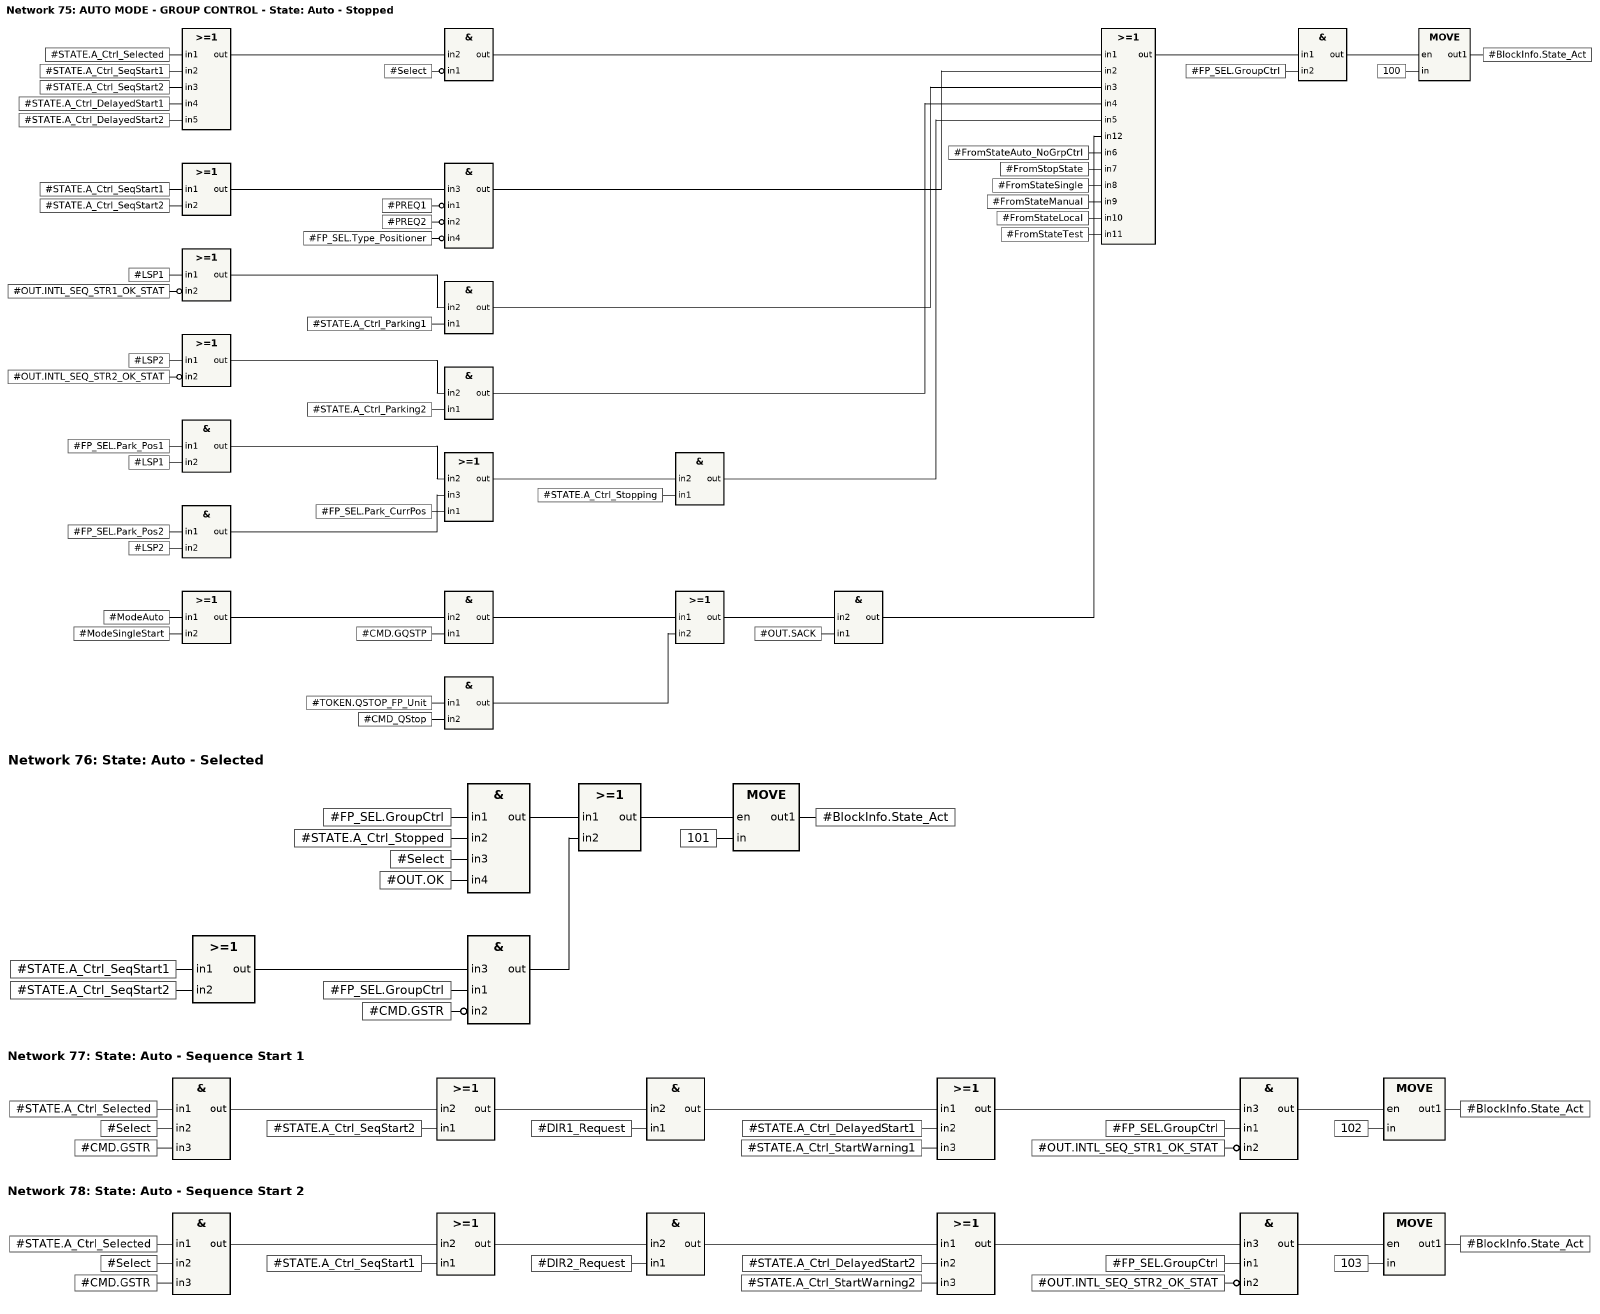
   IF (((#STATE.A_Ctrl_Selected OR #STATE.A_Ctrl_SeqStart1 OR #STATE.A_Ctrl_SeqStart2 OR #STATE.A_Ctrl_DelayedStart1 OR #STATE.A_Ctrl_DelayedStart2) AND NOT #Select) OR ((#STATE.A_Ctrl_SeqStart1 OR #STATE.A_Ctrl_SeqStart2) AND NOT #PREQ1 AND NOT #PREQ2 AND NOT #FP_SEL.Type_Positioner) OR ((#LSP1 OR NOT #OUT.INTL_SEQ_STR1_OK_STAT) AND #STATE.A_Ctrl_Parking1) OR ((#LSP2 OR NOT #OUT.INTL_SEQ_STR2_OK_STAT) AND #STATE.A_Ctrl_Parking2) OR (((#FP_SEL.Park_Pos1 AND #LSP1) OR (#FP_SEL.Park_Pos2 AND #LSP2) OR #FP_SEL.Park_CurrPos) AND #STATE.A_Ctrl_Stopping) OR ((((#ModeAuto OR #ModeSingleStart) AND #CMD.GQSTP) OR (#TOKEN.QSTOP_FP_Unit AND #CMD_QStop)) AND #OUT.SACK) OR #FromStateAuto_NoGrpCtrl OR #FromStopState OR #FromStateSingle OR #FromStateManual OR #FromStateLocal OR #FromStateTest) AND #FP_SEL.GroupCtrl THEN
       #BlockInfo.State_Act := 100;
   END_IF;
END_REGION

REGION Network 76: State: Auto - Selected
   IF (#FP_SEL.GroupCtrl AND #STATE.A_Ctrl_Stopped AND #Select AND #OUT.OK) OR ((#STATE.A_Ctrl_SeqStart1 OR #STATE.A_Ctrl_SeqStart2) AND #FP_SEL.GroupCtrl AND NOT #CMD.GSTR) THEN
       #BlockInfo.State_Act := 101;
   END_IF;
END_REGION

REGION Network 77: State: Auto - Sequence Start 1
   IF ((((#STATE.A_Ctrl_Selected AND #Select AND #CMD.GSTR) OR #STATE.A_Ctrl_SeqStart2) AND #DIR1_Request) OR #STATE.A_Ctrl_DelayedStart1 OR #STATE.A_Ctrl_StartWarning1) AND #FP_SEL.GroupCtrl AND NOT #OUT.INTL_SEQ_STR1_OK_STAT THEN
       #BlockInfo.State_Act := 102;
   END_IF;
END_REGION

REGION Network 78: State: Auto - Sequence Start 2
   IF ((((#STATE.A_Ctrl_Selected AND #Select AND #CMD.GSTR) OR #STATE.A_Ctrl_SeqStart1) AND #DIR2_Request) OR #STATE.A_Ctrl_DelayedStart2 OR #STATE.A_Ctrl_StartWarning2) AND #FP_SEL.GroupCtrl AND NOT #OUT.INTL_SEQ_STR2_OK_STAT THEN
       #BlockInfo.State_Act := 103;
   END_IF;
END_REGION

REGION Network 79: State: Auto - Delayed Start 1
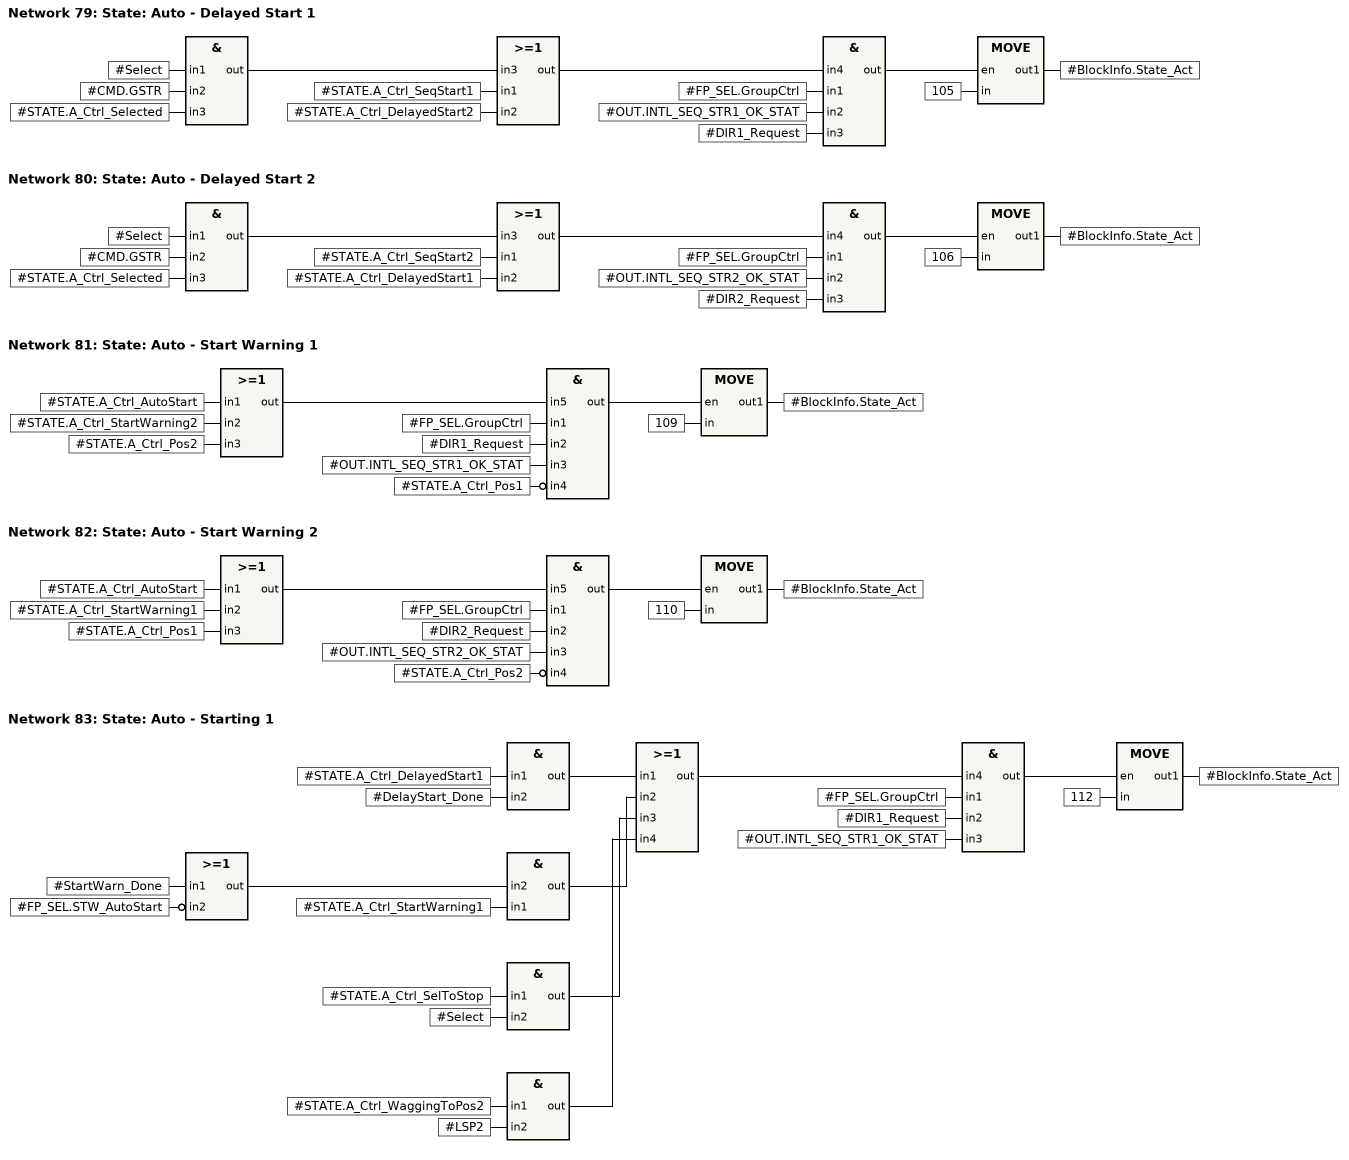
   IF ((#Select AND #CMD.GSTR AND #STATE.A_Ctrl_Selected) OR #STATE.A_Ctrl_SeqStart1 OR #STATE.A_Ctrl_DelayedStart2) AND #FP_SEL.GroupCtrl AND #OUT.INTL_SEQ_STR1_OK_STAT AND #DIR1_Request THEN
       #BlockInfo.State_Act := 105;
   END_IF;
END_REGION

REGION Network 80: State: Auto - Delayed Start 2
   IF ((#Select AND #CMD.GSTR AND #STATE.A_Ctrl_Selected) OR #STATE.A_Ctrl_SeqStart2 OR #STATE.A_Ctrl_DelayedStart1) AND #FP_SEL.GroupCtrl AND #OUT.INTL_SEQ_STR2_OK_STAT AND #DIR2_Request THEN
       #BlockInfo.State_Act := 106;
   END_IF;
END_REGION

REGION Network 81: State: Auto - Start Warning 1
   IF (#STATE.A_Ctrl_AutoStart OR #STATE.A_Ctrl_StartWarning2 OR #STATE.A_Ctrl_Pos2) AND #FP_SEL.GroupCtrl AND #DIR1_Request AND #OUT.INTL_SEQ_STR1_OK_STAT AND NOT #STATE.A_Ctrl_Pos1 THEN
       #BlockInfo.State_Act := 109;
   END_IF;
END_REGION

REGION Network 82: State: Auto - Start Warning 2
   IF (#STATE.A_Ctrl_AutoStart OR #STATE.A_Ctrl_StartWarning1 OR #STATE.A_Ctrl_Pos1) AND #FP_SEL.GroupCtrl AND #DIR2_Request AND #OUT.INTL_SEQ_STR2_OK_STAT AND NOT #STATE.A_Ctrl_Pos2 THEN
       #BlockInfo.State_Act := 110;
   END_IF;
END_REGION

REGION Network 83: State: Auto - Starting 1
   IF ((#STATE.A_Ctrl_DelayedStart1 AND #DelayStart_Done) OR ((#StartWarn_Done OR NOT #FP_SEL.STW_AutoStart) AND #STATE.A_Ctrl_StartWarning1) OR (#STATE.A_Ctrl_SelToStop AND #Select) OR (#STATE.A_Ctrl_WaggingToPos2 AND #LSP2)) AND #FP_SEL.GroupCtrl AND #DIR1_Request AND #OUT.INTL_SEQ_STR1_OK_STAT THEN
       #BlockInfo.State_Act := 112;
   END_IF;
END_REGION

REGION Network 84: state: Auto - Starting 2
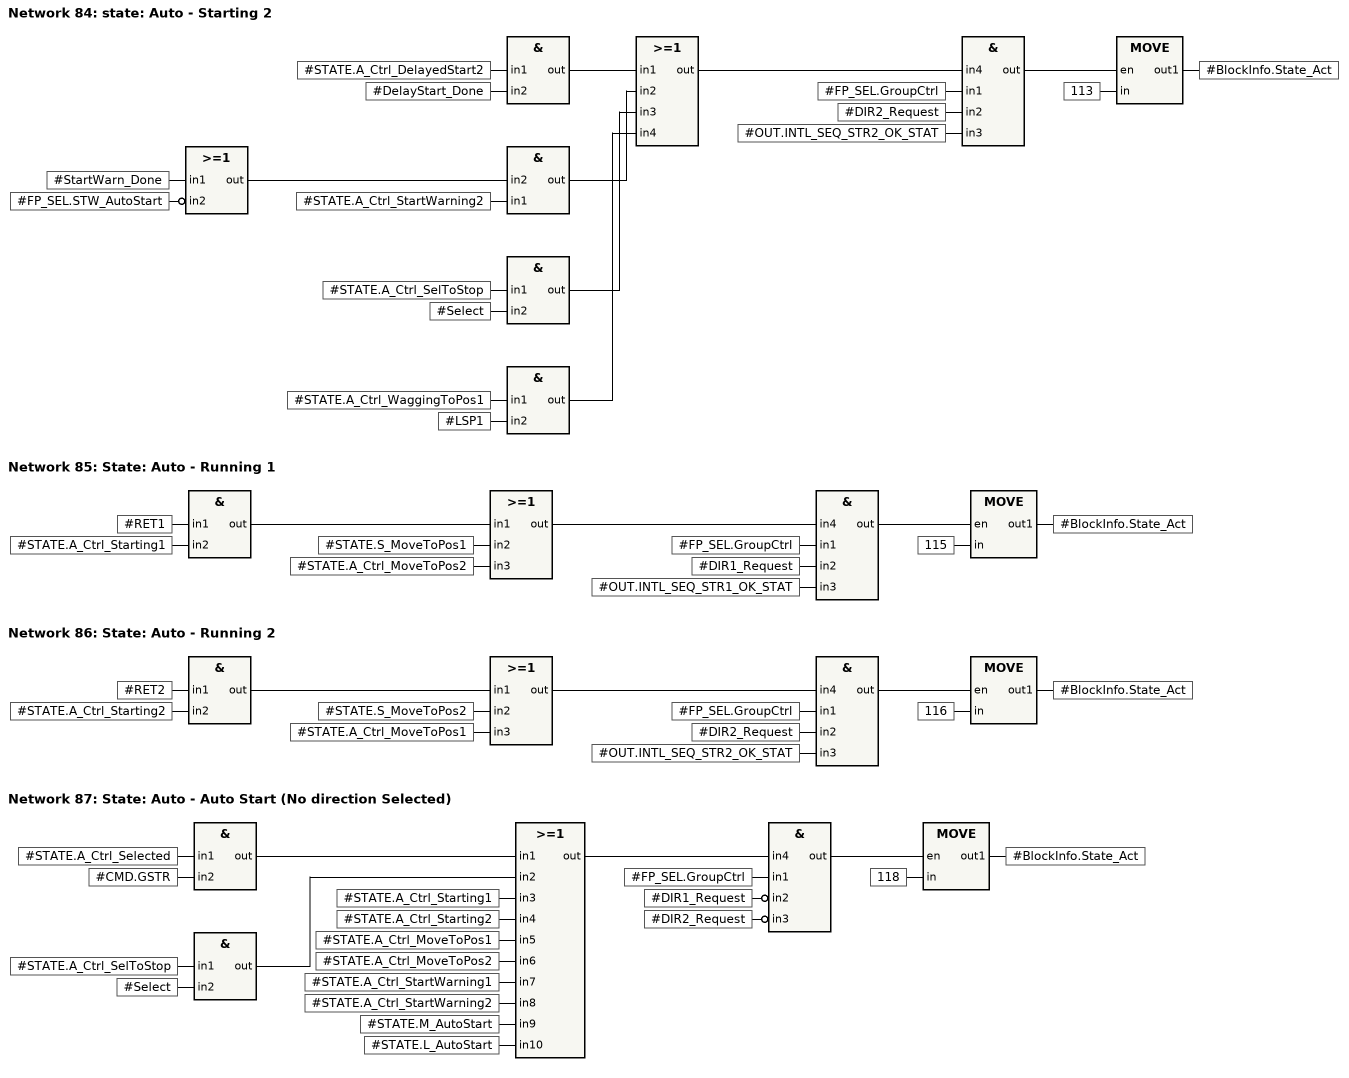
   IF ((#STATE.A_Ctrl_DelayedStart2 AND #DelayStart_Done) OR ((#StartWarn_Done OR NOT #FP_SEL.STW_AutoStart) AND #STATE.A_Ctrl_StartWarning2) OR (#STATE.A_Ctrl_SelToStop AND #Select) OR (#STATE.A_Ctrl_WaggingToPos1 AND #LSP1)) AND #FP_SEL.GroupCtrl AND #DIR2_Request AND #OUT.INTL_SEQ_STR2_OK_STAT THEN
       #BlockInfo.State_Act := 113;
   END_IF;
END_REGION

REGION Network 85: State: Auto - Running 1
   IF ((#RET1 AND #STATE.A_Ctrl_Starting1) OR #STATE.S_MoveToPos1 OR #STATE.A_Ctrl_MoveToPos2) AND #FP_SEL.GroupCtrl AND #DIR1_Request AND #OUT.INTL_SEQ_STR1_OK_STAT THEN
       #BlockInfo.State_Act := 115;
   END_IF;
END_REGION

REGION Network 86: State: Auto - Running 2
   IF ((#RET2 AND #STATE.A_Ctrl_Starting2) OR #STATE.S_MoveToPos2 OR #STATE.A_Ctrl_MoveToPos1) AND #FP_SEL.GroupCtrl AND #DIR2_Request AND #OUT.INTL_SEQ_STR2_OK_STAT THEN
       #BlockInfo.State_Act := 116;
   END_IF;
END_REGION

REGION Network 87: State: Auto - Auto Start (No direction Selected)
   // Build 002 - 26 March 2019 : SetToStop with Select condition is added
   IF ((#STATE.A_Ctrl_Selected AND #CMD.GSTR) OR (#STATE.A_Ctrl_SelToStop AND #Select) OR #STATE.A_Ctrl_Starting1 OR #STATE.A_Ctrl_Starting2 OR #STATE.A_Ctrl_MoveToPos1 OR #STATE.A_Ctrl_MoveToPos2 OR #STATE.A_Ctrl_StartWarning1 OR #STATE.A_Ctrl_StartWarning2 OR #STATE.M_AutoStart OR #STATE.L_AutoStart) AND #FP_SEL.GroupCtrl AND NOT #DIR1_Request AND NOT #DIR2_Request THEN
       #BlockInfo.State_Act := 118;
   END_IF;
END_REGION

REGION Network 88: State: Auto - In Pos. 1
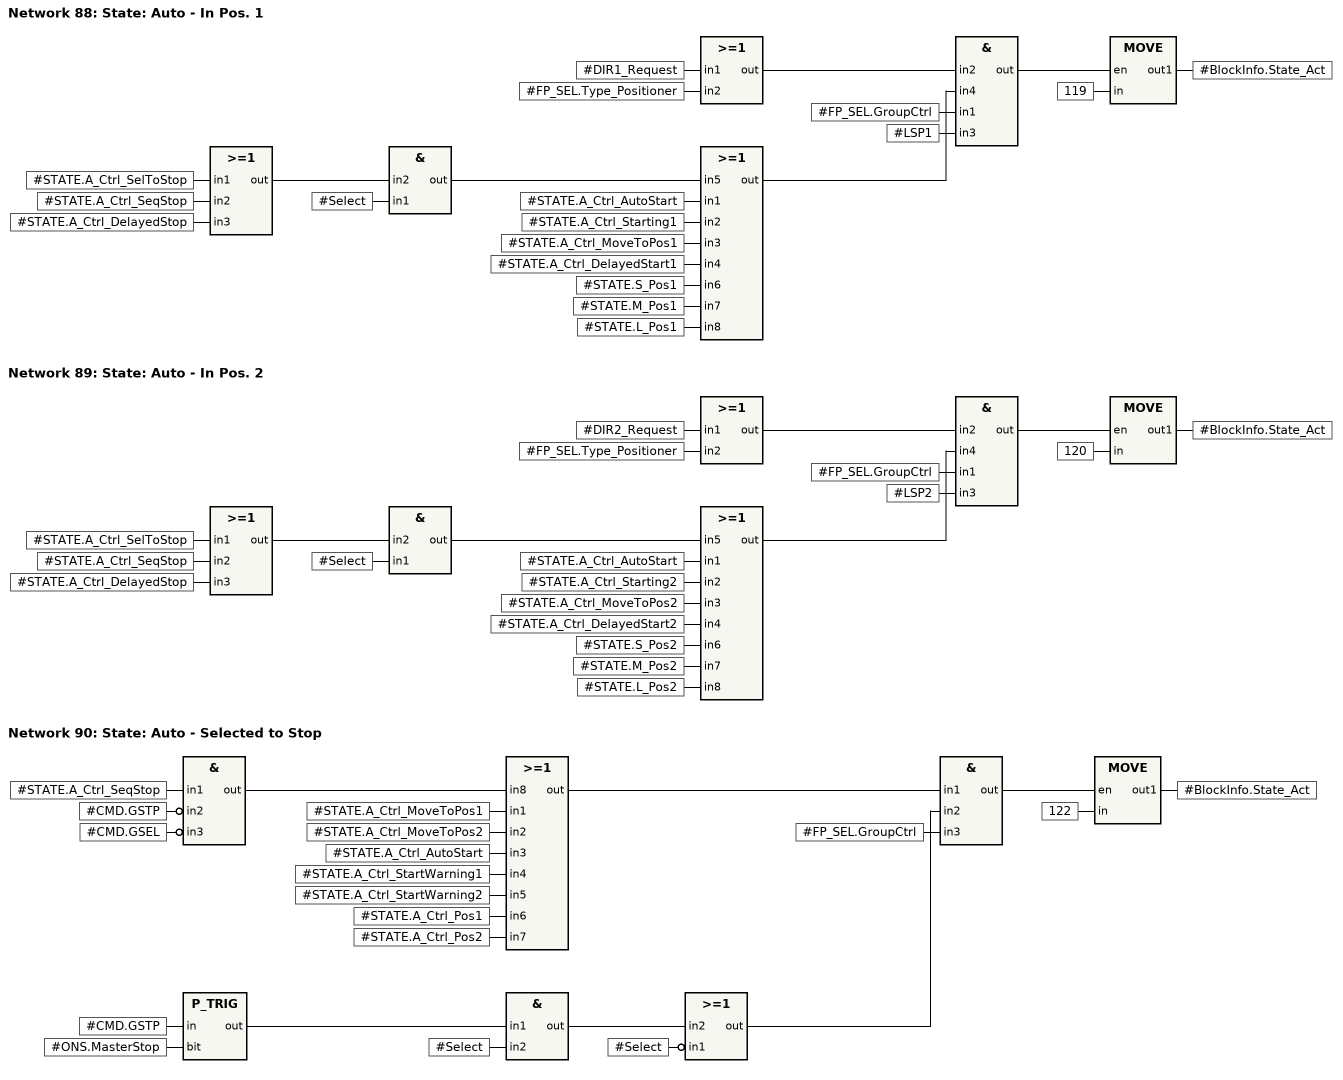
   IF (#DIR1_Request OR #FP_SEL.Type_Positioner) AND (((#STATE.A_Ctrl_SelToStop OR #STATE.A_Ctrl_SeqStop OR #STATE.A_Ctrl_DelayedStop) AND #Select) OR #STATE.A_Ctrl_AutoStart OR #STATE.A_Ctrl_Starting1 OR #STATE.A_Ctrl_MoveToPos1 OR #STATE.A_Ctrl_DelayedStart1 OR #STATE.S_Pos1 OR #STATE.M_Pos1 OR #STATE.L_Pos1) AND #FP_SEL.GroupCtrl AND #LSP1 THEN
       #BlockInfo.State_Act := 119;
   END_IF;
END_REGION

REGION Network 89: State: Auto - In Pos. 2
   IF (#DIR2_Request OR #FP_SEL.Type_Positioner) AND (((#STATE.A_Ctrl_SelToStop OR #STATE.A_Ctrl_SeqStop OR #STATE.A_Ctrl_DelayedStop) AND #Select) OR #STATE.A_Ctrl_AutoStart OR #STATE.A_Ctrl_Starting2 OR #STATE.A_Ctrl_MoveToPos2 OR #STATE.A_Ctrl_DelayedStart2 OR #STATE.S_Pos2 OR #STATE.M_Pos2 OR #STATE.L_Pos2) AND #FP_SEL.GroupCtrl AND #LSP2 THEN
       #BlockInfo.State_Act := 120;
   END_IF;
END_REGION

REGION Network 90: State: Auto - Selected to Stop
   // Build 004 - 11 Jul 2019 (EXTBOB) : GSEL and A_Ctrl_SeqStop with GSTP condition to move to Selected to Stop state from Seq stop state if group stop timer completes
   #_w1 := #CMD.GSTP AND NOT #ONS.MasterStop;   // rising edge
   #ONS.MasterStop := #CMD.GSTP;
   IF ((#STATE.A_Ctrl_SeqStop AND NOT #CMD.GSTP AND NOT #CMD.GSEL) OR #STATE.A_Ctrl_MoveToPos1 OR #STATE.A_Ctrl_MoveToPos2 OR #STATE.A_Ctrl_AutoStart OR #STATE.A_Ctrl_StartWarning1 OR #STATE.A_Ctrl_StartWarning2 OR #STATE.A_Ctrl_Pos1 OR #STATE.A_Ctrl_Pos2) AND ((#_w1 AND #Select) OR NOT #Select) AND #FP_SEL.GroupCtrl THEN
       #BlockInfo.State_Act := 122;
   END_IF;
END_REGION

REGION Network 91: State: Auto - Sequence Stop
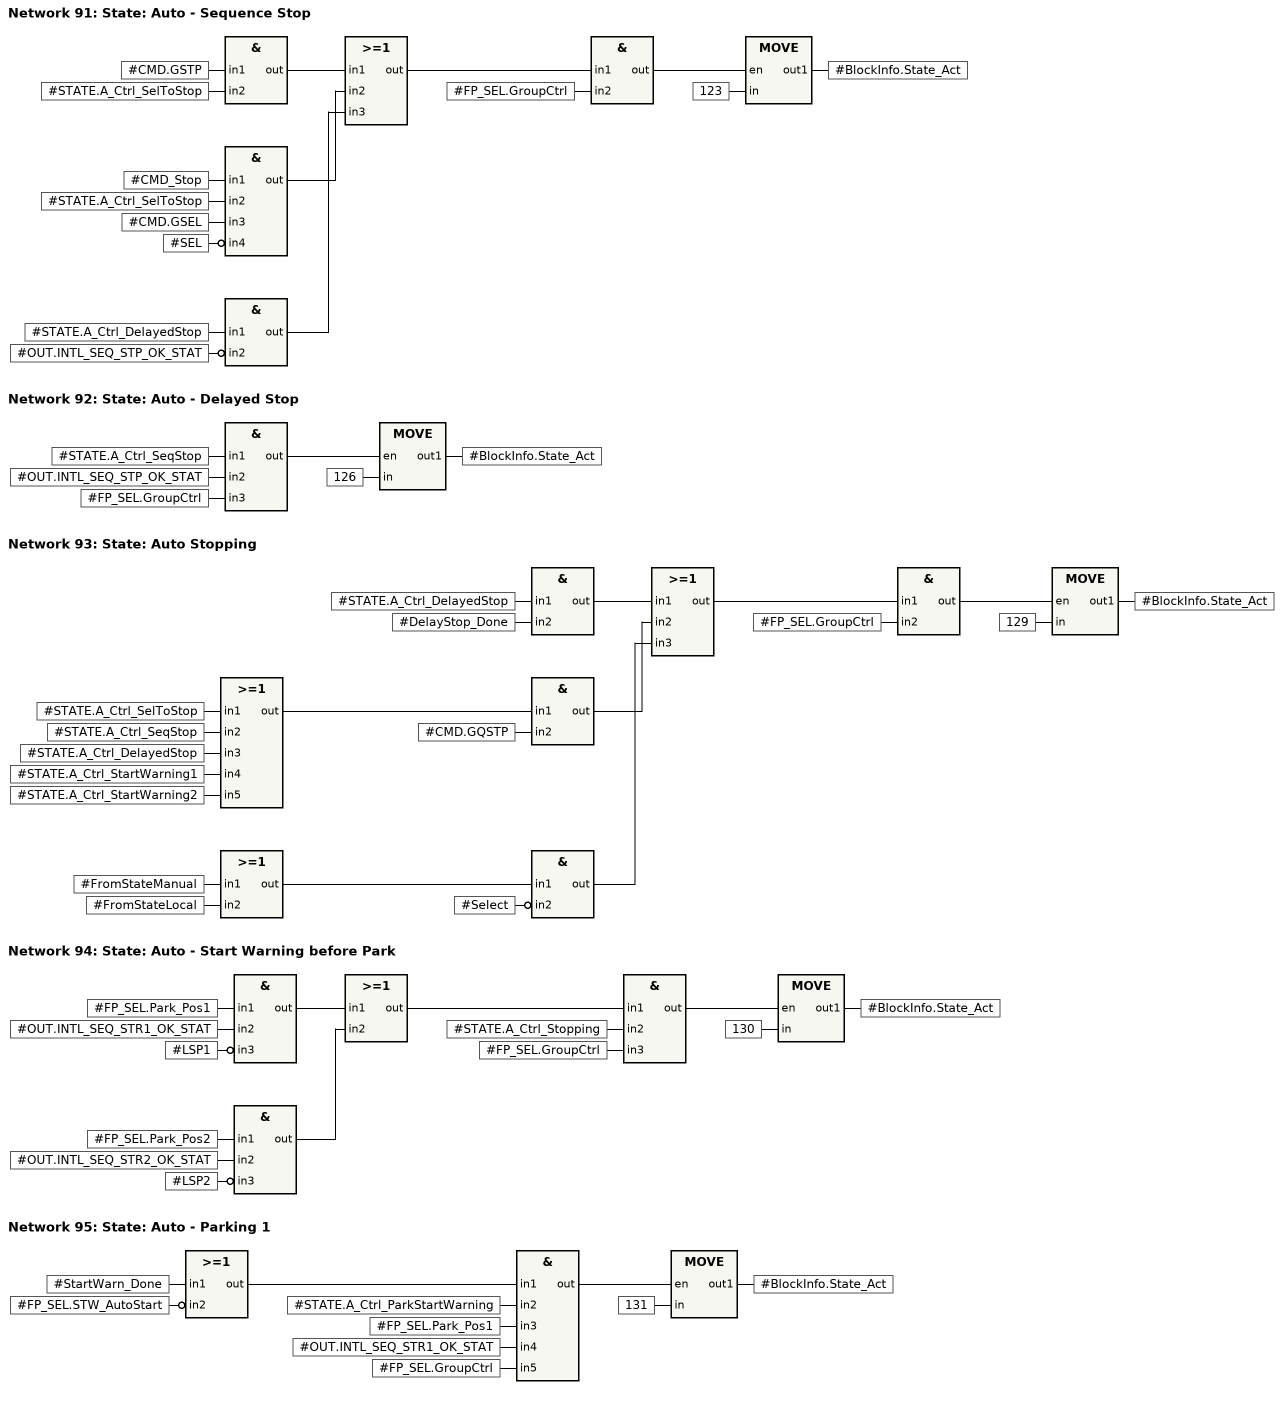
   IF ((#CMD.GSTP AND #STATE.A_Ctrl_SelToStop) OR (#CMD_Stop AND #STATE.A_Ctrl_SelToStop AND #CMD.GSEL AND NOT #SEL) OR (#STATE.A_Ctrl_DelayedStop AND NOT #OUT.INTL_SEQ_STP_OK_STAT)) AND #FP_SEL.GroupCtrl THEN
       #BlockInfo.State_Act := 123;
   END_IF;
END_REGION

REGION Network 92: State: Auto - Delayed Stop
   IF #STATE.A_Ctrl_SeqStop AND #OUT.INTL_SEQ_STP_OK_STAT AND #FP_SEL.GroupCtrl THEN
       #BlockInfo.State_Act := 126;
   END_IF;
END_REGION

REGION Network 93: State: Auto Stopping
   IF ((#STATE.A_Ctrl_DelayedStop AND #DelayStop_Done) OR ((#STATE.A_Ctrl_SelToStop OR #STATE.A_Ctrl_SeqStop OR #STATE.A_Ctrl_DelayedStop OR #STATE.A_Ctrl_StartWarning1 OR #STATE.A_Ctrl_StartWarning2) AND #CMD.GQSTP) OR ((#FromStateManual OR #FromStateLocal) AND NOT #Select)) AND #FP_SEL.GroupCtrl THEN
       #BlockInfo.State_Act := 129;
   END_IF;
END_REGION

REGION Network 94: State: Auto - Start Warning before Park
   IF ((#FP_SEL.Park_Pos1 AND #OUT.INTL_SEQ_STR1_OK_STAT AND NOT #LSP1) OR (#FP_SEL.Park_Pos2 AND #OUT.INTL_SEQ_STR2_OK_STAT AND NOT #LSP2)) AND #STATE.A_Ctrl_Stopping AND #FP_SEL.GroupCtrl THEN
       #BlockInfo.State_Act := 130;
   END_IF;
END_REGION

REGION Network 95: State: Auto - Parking 1
   IF (#StartWarn_Done OR NOT #FP_SEL.STW_AutoStart) AND #STATE.A_Ctrl_ParkStartWarning AND #FP_SEL.Park_Pos1 AND #OUT.INTL_SEQ_STR1_OK_STAT AND #FP_SEL.GroupCtrl THEN
       #BlockInfo.State_Act := 131;
   END_IF;
END_REGION

REGION Network 96: State: Auto - Parking 2
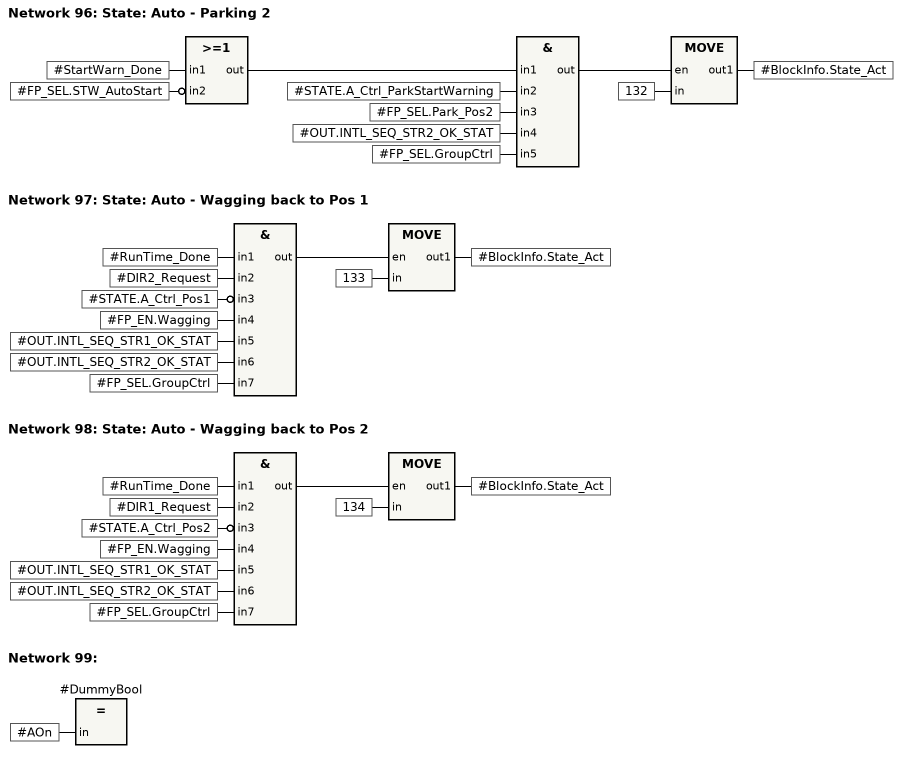
   IF (#StartWarn_Done OR NOT #FP_SEL.STW_AutoStart) AND #STATE.A_Ctrl_ParkStartWarning AND #FP_SEL.Park_Pos2 AND #OUT.INTL_SEQ_STR2_OK_STAT AND #FP_SEL.GroupCtrl THEN
       #BlockInfo.State_Act := 132;
   END_IF;
END_REGION

REGION Network 97: State: Auto - Wagging back to Pos 1
   IF #RunTime_Done AND #DIR2_Request AND NOT #STATE.A_Ctrl_Pos1 AND #FP_EN.Wagging AND #OUT.INTL_SEQ_STR1_OK_STAT AND #OUT.INTL_SEQ_STR2_OK_STAT AND #FP_SEL.GroupCtrl THEN
       #BlockInfo.State_Act := 133;
   END_IF;
END_REGION

REGION Network 98: State: Auto - Wagging back to Pos 2
   IF #RunTime_Done AND #DIR1_Request AND NOT #STATE.A_Ctrl_Pos2 AND #FP_EN.Wagging AND #OUT.INTL_SEQ_STR1_OK_STAT AND #OUT.INTL_SEQ_STR2_OK_STAT AND #FP_SEL.GroupCtrl THEN
       #BlockInfo.State_Act := 134;
   END_IF;
END_REGION

REGION Network 99
   INDC:
   #DummyBool := #AOn;
END_REGION

REGION Network 100: AUTO MODE - NO GROUP CONTROL
   // State: Auto - Auto Start (No direction Selected)
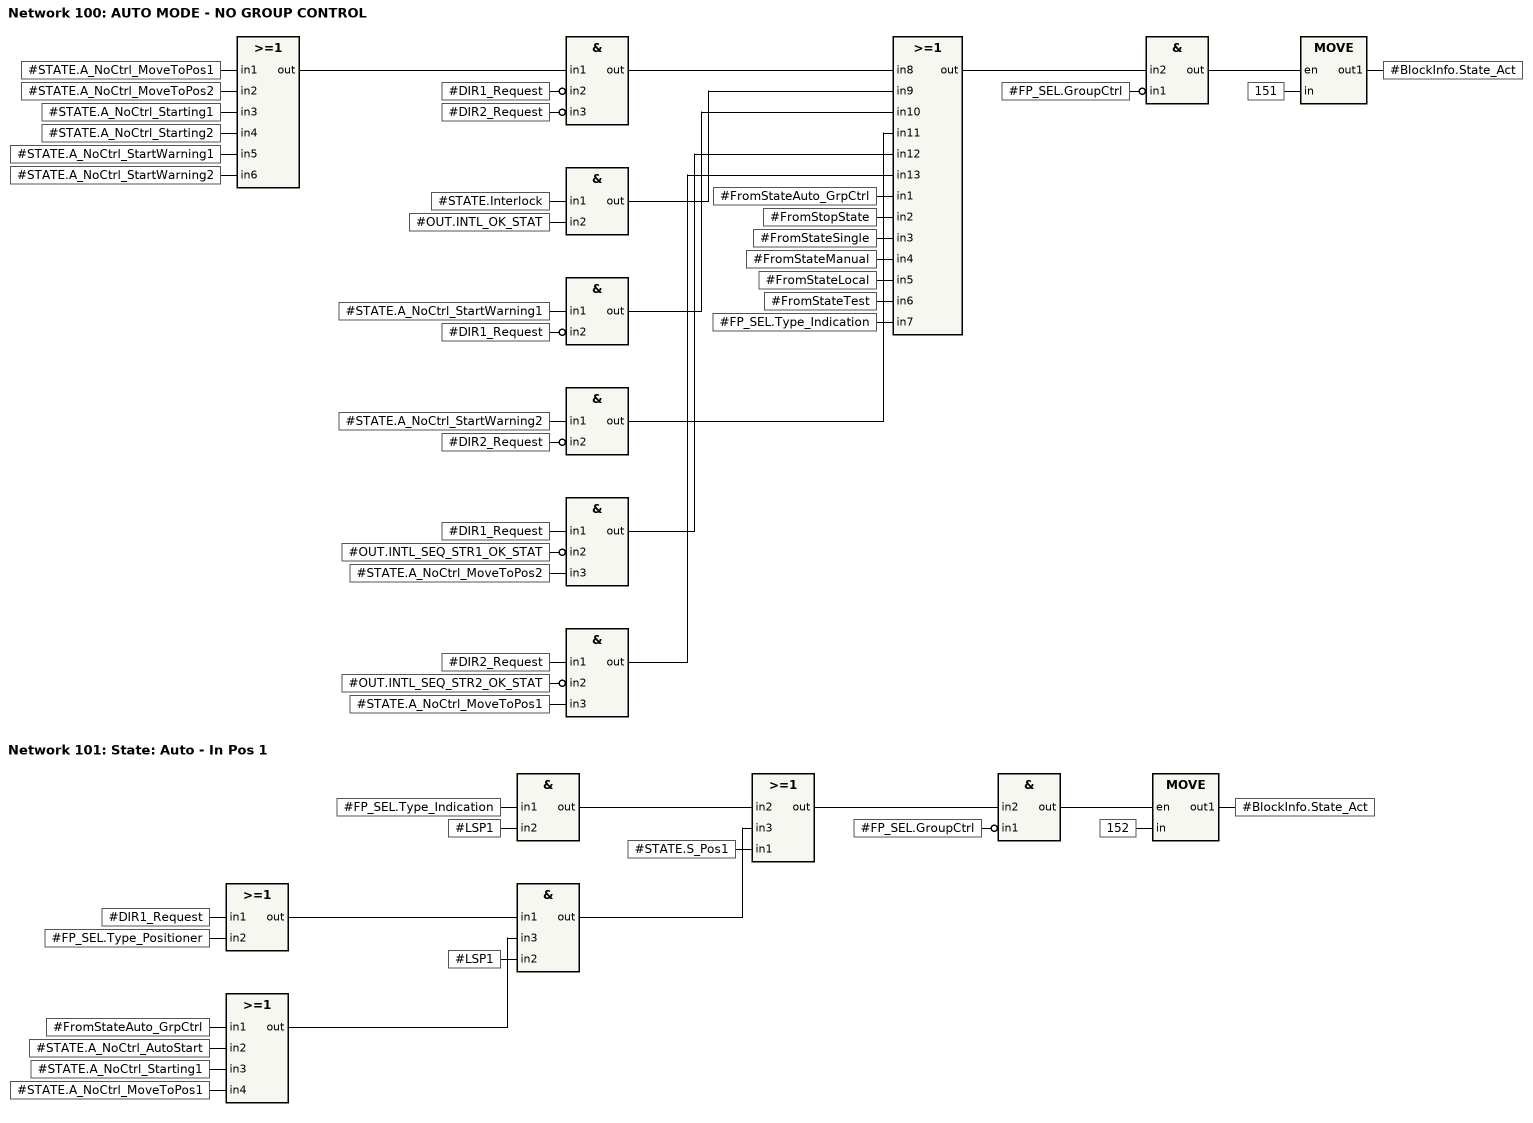
   IF (((#STATE.A_NoCtrl_MoveToPos1 OR #STATE.A_NoCtrl_MoveToPos2 OR #STATE.A_NoCtrl_Starting1 OR #STATE.A_NoCtrl_Starting2 OR #STATE.A_NoCtrl_StartWarning1 OR #STATE.A_NoCtrl_StartWarning2) AND NOT #DIR1_Request AND NOT #DIR2_Request) OR (#STATE.Interlock AND #OUT.INTL_OK_STAT) OR (#STATE.A_NoCtrl_StartWarning1 AND NOT #DIR1_Request) OR (#STATE.A_NoCtrl_StartWarning2 AND NOT #DIR2_Request) OR (#DIR1_Request AND NOT #OUT.INTL_SEQ_STR1_OK_STAT AND #STATE.A_NoCtrl_MoveToPos2) OR (#DIR2_Request AND NOT #OUT.INTL_SEQ_STR2_OK_STAT AND #STATE.A_NoCtrl_MoveToPos1) OR #FromStateAuto_GrpCtrl OR #FromStopState OR #FromStateSingle OR #FromStateManual OR #FromStateLocal OR #FromStateTest OR #FP_SEL.Type_Indication) AND NOT #FP_SEL.GroupCtrl THEN
       #BlockInfo.State_Act := 151;
   END_IF;
END_REGION

REGION Network 101: State: Auto - In Pos 1
   IF ((#FP_SEL.Type_Indication AND #LSP1) OR ((#DIR1_Request OR #FP_SEL.Type_Positioner) AND (#FromStateAuto_GrpCtrl OR #STATE.A_NoCtrl_AutoStart OR #STATE.A_NoCtrl_Starting1 OR #STATE.A_NoCtrl_MoveToPos1) AND #LSP1) OR #STATE.S_Pos1) AND NOT #FP_SEL.GroupCtrl THEN
       #BlockInfo.State_Act := 152;
   END_IF;
END_REGION

REGION Network 102: State: Auto - In Pos 2
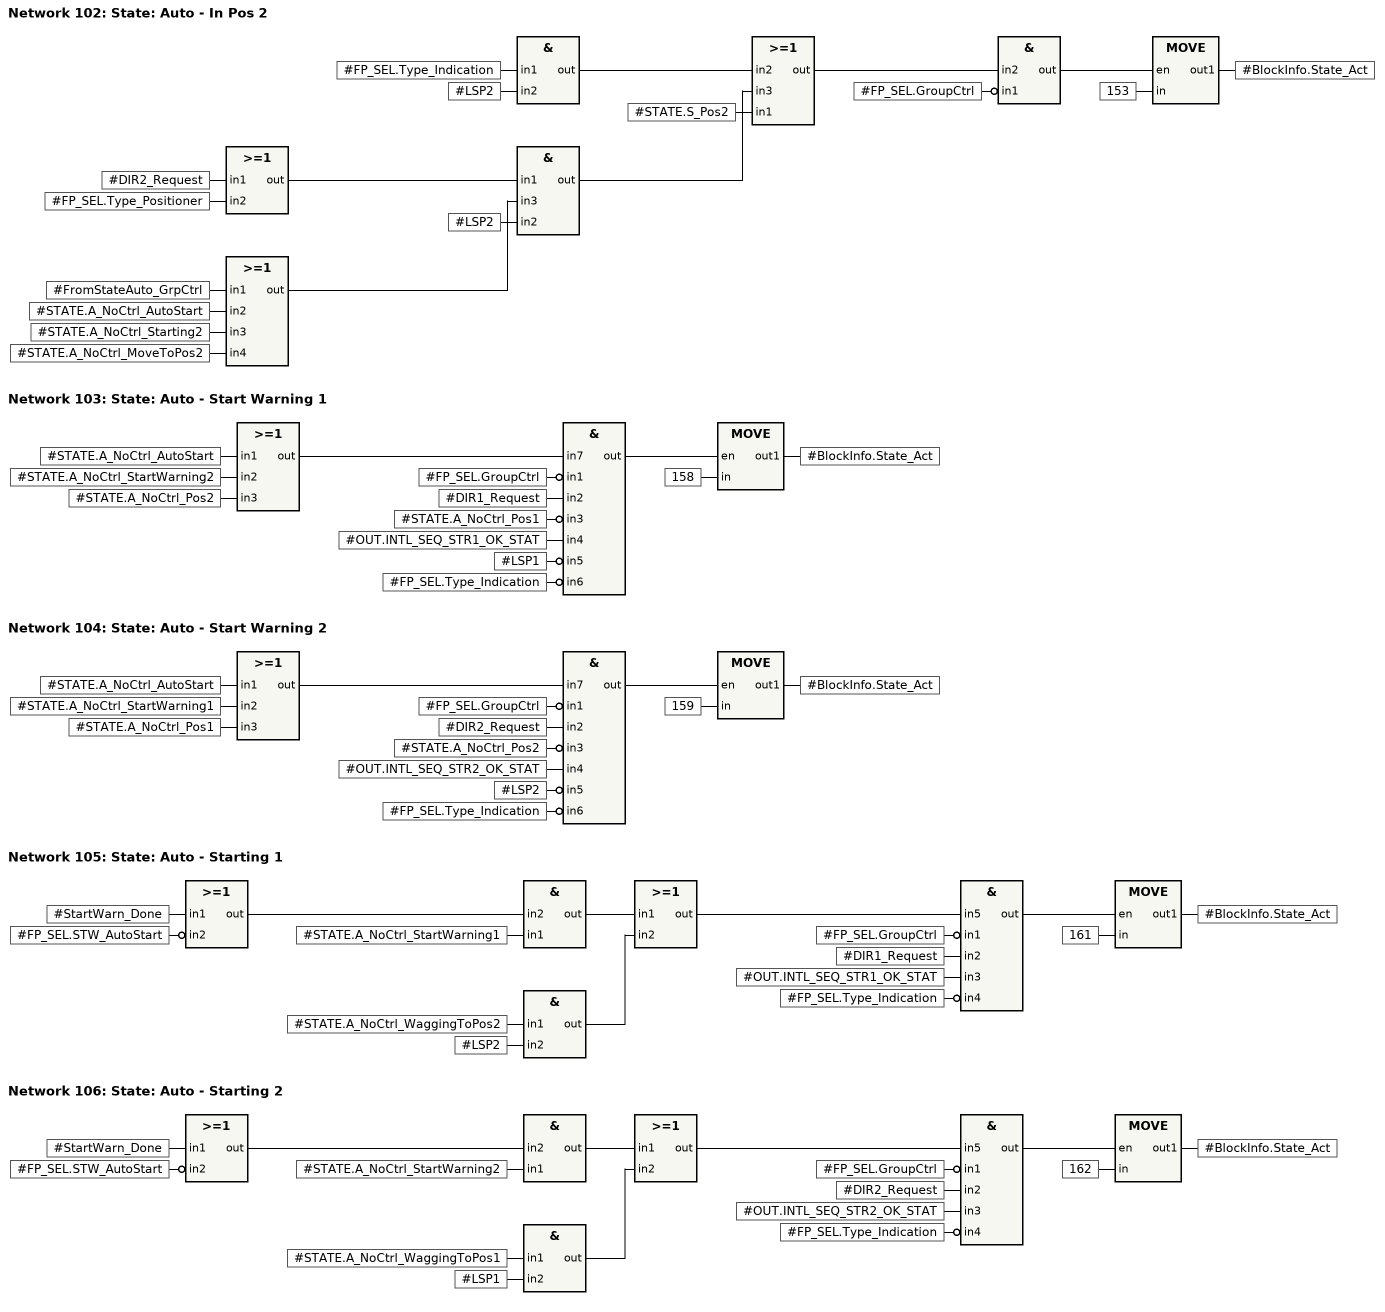
   IF ((#FP_SEL.Type_Indication AND #LSP2) OR ((#DIR2_Request OR #FP_SEL.Type_Positioner) AND (#FromStateAuto_GrpCtrl OR #STATE.A_NoCtrl_AutoStart OR #STATE.A_NoCtrl_Starting2 OR #STATE.A_NoCtrl_MoveToPos2) AND #LSP2) OR #STATE.S_Pos2) AND NOT #FP_SEL.GroupCtrl THEN
       #BlockInfo.State_Act := 153;
   END_IF;
END_REGION

REGION Network 103: State: Auto - Start Warning 1
   IF (#STATE.A_NoCtrl_AutoStart OR #STATE.A_NoCtrl_StartWarning2 OR #STATE.A_NoCtrl_Pos2) AND NOT #FP_SEL.GroupCtrl AND #DIR1_Request AND NOT #STATE.A_NoCtrl_Pos1 AND #OUT.INTL_SEQ_STR1_OK_STAT AND NOT #LSP1 AND NOT #FP_SEL.Type_Indication THEN
       #BlockInfo.State_Act := 158;
   END_IF;
END_REGION

REGION Network 104: State: Auto - Start Warning 2
   IF (#STATE.A_NoCtrl_AutoStart OR #STATE.A_NoCtrl_StartWarning1 OR #STATE.A_NoCtrl_Pos1) AND NOT #FP_SEL.GroupCtrl AND #DIR2_Request AND NOT #STATE.A_NoCtrl_Pos2 AND #OUT.INTL_SEQ_STR2_OK_STAT AND NOT #LSP2 AND NOT #FP_SEL.Type_Indication THEN
       #BlockInfo.State_Act := 159;
   END_IF;
END_REGION

REGION Network 105: State: Auto - Starting 1
   IF (((#StartWarn_Done OR NOT #FP_SEL.STW_AutoStart) AND #STATE.A_NoCtrl_StartWarning1) OR (#STATE.A_NoCtrl_WaggingToPos2 AND #LSP2)) AND NOT #FP_SEL.GroupCtrl AND #DIR1_Request AND #OUT.INTL_SEQ_STR1_OK_STAT AND NOT #FP_SEL.Type_Indication THEN
       #BlockInfo.State_Act := 161;
   END_IF;
END_REGION

REGION Network 106: State: Auto - Starting 2
   IF (((#StartWarn_Done OR NOT #FP_SEL.STW_AutoStart) AND #STATE.A_NoCtrl_StartWarning2) OR (#STATE.A_NoCtrl_WaggingToPos1 AND #LSP1)) AND NOT #FP_SEL.GroupCtrl AND #DIR2_Request AND #OUT.INTL_SEQ_STR2_OK_STAT AND NOT #FP_SEL.Type_Indication THEN
       #BlockInfo.State_Act := 162;
   END_IF;
END_REGION

REGION Network 107: State: Auto - Running 1
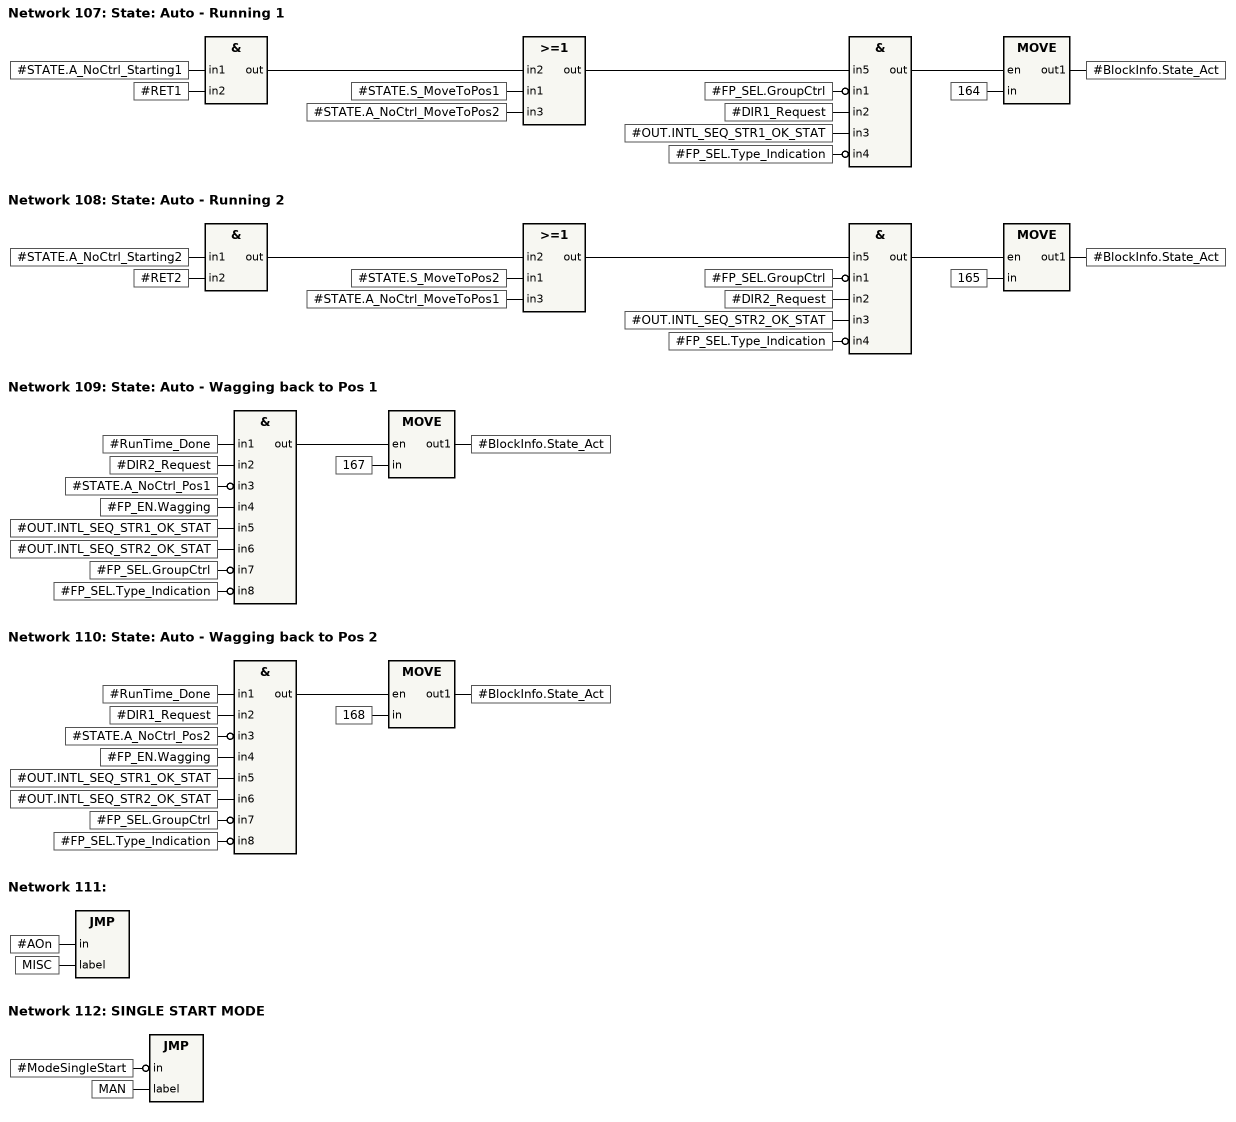
   IF ((#STATE.A_NoCtrl_Starting1 AND #RET1) OR #STATE.S_MoveToPos1 OR #STATE.A_NoCtrl_MoveToPos2) AND NOT #FP_SEL.GroupCtrl AND #DIR1_Request AND #OUT.INTL_SEQ_STR1_OK_STAT AND NOT #FP_SEL.Type_Indication THEN
       #BlockInfo.State_Act := 164;
   END_IF;
END_REGION

REGION Network 108: State: Auto - Running 2
   IF ((#STATE.A_NoCtrl_Starting2 AND #RET2) OR #STATE.S_MoveToPos2 OR #STATE.A_NoCtrl_MoveToPos1) AND NOT #FP_SEL.GroupCtrl AND #DIR2_Request AND #OUT.INTL_SEQ_STR2_OK_STAT AND NOT #FP_SEL.Type_Indication THEN
       #BlockInfo.State_Act := 165;
   END_IF;
END_REGION

REGION Network 109: State: Auto - Wagging back to Pos 1
   IF #RunTime_Done AND #DIR2_Request AND NOT #STATE.A_NoCtrl_Pos1 AND #FP_EN.Wagging AND #OUT.INTL_SEQ_STR1_OK_STAT AND #OUT.INTL_SEQ_STR2_OK_STAT AND NOT #FP_SEL.GroupCtrl AND NOT #FP_SEL.Type_Indication THEN
       #BlockInfo.State_Act := 167;
   END_IF;
END_REGION

REGION Network 110: State: Auto - Wagging back to Pos 2
   IF #RunTime_Done AND #DIR1_Request AND NOT #STATE.A_NoCtrl_Pos2 AND #FP_EN.Wagging AND #OUT.INTL_SEQ_STR1_OK_STAT AND #OUT.INTL_SEQ_STR2_OK_STAT AND NOT #FP_SEL.GroupCtrl AND NOT #FP_SEL.Type_Indication THEN
       #BlockInfo.State_Act := 168;
   END_IF;
END_REGION

REGION Network 111
   IF #AOn THEN GOTO MISC; END_IF;
END_REGION

REGION Network 112: SINGLE START MODE
   SS1:
   IF NOT #ModeSingleStart THEN GOTO MAN; END_IF;
END_REGION

REGION Network 113: State: Single Start - Not Active
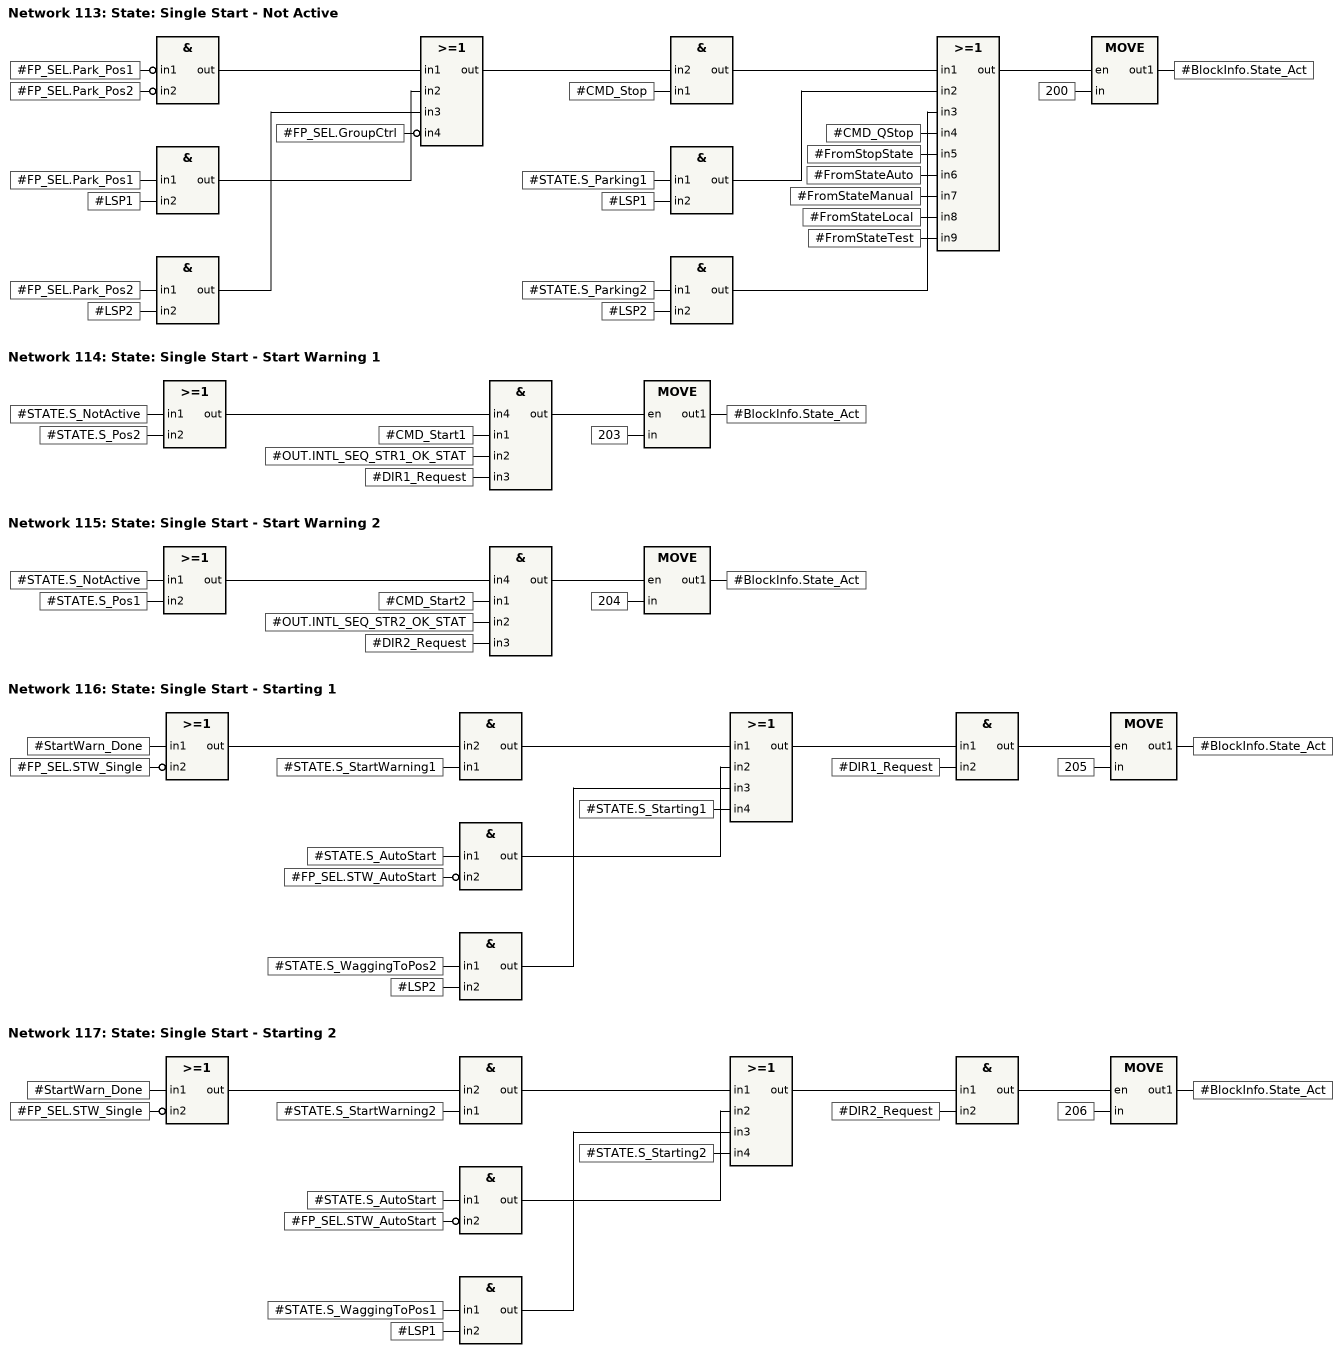
   IF (((NOT #FP_SEL.Park_Pos1 AND NOT #FP_SEL.Park_Pos2) OR (#FP_SEL.Park_Pos1 AND #LSP1) OR (#FP_SEL.Park_Pos2 AND #LSP2) OR NOT #FP_SEL.GroupCtrl) AND #CMD_Stop) OR (#STATE.S_Parking1 AND #LSP1) OR (#STATE.S_Parking2 AND #LSP2) OR #CMD_QStop OR #FromStopState OR #FromStateAuto OR #FromStateManual OR #FromStateLocal OR #FromStateTest THEN
       #BlockInfo.State_Act := 200;
   END_IF;
END_REGION

REGION Network 114: State: Single Start - Start Warning 1
   IF (#STATE.S_NotActive OR #STATE.S_Pos2) AND #CMD_Start1 AND #OUT.INTL_SEQ_STR1_OK_STAT AND #DIR1_Request THEN
       #BlockInfo.State_Act := 203;
   END_IF;
END_REGION

REGION Network 115: State: Single Start - Start Warning 2
   IF (#STATE.S_NotActive OR #STATE.S_Pos1) AND #CMD_Start2 AND #OUT.INTL_SEQ_STR2_OK_STAT AND #DIR2_Request THEN
       #BlockInfo.State_Act := 204;
   END_IF;
END_REGION

REGION Network 116: State: Single Start - Starting 1
   IF (((#StartWarn_Done OR NOT #FP_SEL.STW_Single) AND #STATE.S_StartWarning1) OR (#STATE.S_AutoStart AND NOT #FP_SEL.STW_AutoStart) OR (#STATE.S_WaggingToPos2 AND #LSP2) OR #STATE.S_Starting1) AND #DIR1_Request THEN
       #BlockInfo.State_Act := 205;
   END_IF;
END_REGION

REGION Network 117: State: Single Start - Starting 2
   IF (((#StartWarn_Done OR NOT #FP_SEL.STW_Single) AND #STATE.S_StartWarning2) OR (#STATE.S_AutoStart AND NOT #FP_SEL.STW_AutoStart) OR (#STATE.S_WaggingToPos1 AND #LSP1) OR #STATE.S_Starting2) AND #DIR2_Request THEN
       #BlockInfo.State_Act := 206;
   END_IF;
END_REGION

REGION Network 118: State: Single Start - Running 1
